// TwinCAT 3 PLC project Library
// Title: lcls-twincat-common-components
// Company: SLAC
// ProjectVersion: 0.0.0
// ProgramVersion: 3.1.4026.17
// libraries:
//   LCLS General, * (SLAC)
//   lcls-twincat-motion, * (SLAC)
//   lcls-twincat-physics, * (SLAC)
//   PMPS, * (SLAC - LCLS)
//   Tc2_MC2, * (Beckhoff Automation GmbH)
//   Tc2_SerialCom, * (Beckhoff Automation GmbH)
//   Tc2_Standard, * (Beckhoff Automation GmbH)
//   Tc2_System, * (Beckhoff Automation GmbH)
//   Tc2_Utilities, * (Beckhoff Automation GmbH)
//   Tc3_JsonXml, * (Beckhoff Automation GmbH)
//   Tc3_Module, * (Beckhoff Automation GmbH)
//   TcUnit, * (www.tcunit.org)
// project tree:
//   Devices/ATM/ E_ATM_States.TcDUT (not stored), FB_ATM.TcPOU (not stored)
//   Devices/HE_SATT/ E_HE_SATT_FilterMaterial.TcDUT, E_HE_SATT_FilterStatus.TcDUT, E_HE_SATT_FilterType.TcDUT, E_HE_SATT_RoundingMode.TcDUT, E_HE_SATT_SequenceState.TcDUT, F_HE_SATT_MaterialToMaterialFormula.TcPOU, PL_HE_SATT_Parameters.TcGVL, ST_HE_SATT_Status.TcDUT
//   Devices/HE_SATT/FBs/ FB_HE_SATT.TcPOU, FB_HE_SATT_CommandsEpics.TcPOU, FB_HE_SATT_EpicsHeartBeat.TcPOU, FB_HE_SATT_Filter.TcPOU, FB_HE_SATT_FilterCombination.TcPOU (not stored), FB_HE_SATT_FilterCombinationCollector.TcPOU, FB_HE_SATT_FilterCombinationFinder.TcPOU, FB_HE_SATT_FilterCombinationToTransmission.TcPOU, FB_HE_SATT_FilterConstantThickness.TcPOU, FB_HE_SATT_FilterHolder.TcPOU, FB_HE_SATT_FilterHolderSelector.TcPOU, FB_HE_SATT_FindOptimalFilterCombination.TcPOU, FB_HE_SATT_FilterToTransmission.TcPOU, FB_HE_SATT_FilterWedge.TcPOU, FB_HE_SATT_Sequence.TcPOU, FB_HE_SATT_UserRequest.TcPOU
//   Devices/HE_SATT/ITFs/ I_HE_SATT_Commands.TcIO, I_HE_SATT_Filter.TcIO, I_HE_SATT_FilterCombination.TcIO, I_HE_SATT_FilterCombinationCollector.TcIO, I_HE_SATT_FilterCombinationFinder.TcIO, I_HE_SATT_FilterCombinationToTransmission.TcIO, I_HE_SATT_FilterConstantThickness.TcIO (not stored), I_HE_SATT_FilterHolder.TcIO, I_HE_SATT_FilterHolderSelector.TcIO, I_HE_SATT_FilterToTransmission.TcIO, I_HE_SATT_FilterWedge.TcIO, I_HE_SATT_FindOptimalFilterCombination.TcIO, I_HE_SATT_FindOptimalThicknessFromFilterCombination.TcIO, I_HE_SATT_PhotonEnergy_eV.TcIO, I_HE_SATT_Sequence.TcIO
//   Devices/LIC/ E_LIC_States.TcDUT (not stored), FB_LIC.TcPOU (not stored)
//   Devices/PPM/ E_PPM_States.TcDUT (not stored), FB_PPM.TcPOU (not stored), FB_PPM_Gige.TcPOU (not stored), FB_PPM_PowerMeter.TcPOU
//   Devices/REF/ FB_REF.TcPOU (not stored), FB_REF_Laser.TcPOU (not stored)
//   Devices/SATT/ E_SXR_SATT_Position.TcDUT (not stored), FB_AttenuatorElementDensity.TcPOU (not stored), FB_SXR_SATT_Stage.TcPOU (not stored), ST_SATT_Filter.TcDUT (not stored)
//   Devices/SLITS/ FB_SLITS.TcPOU (not stored), FB_SLITS_POWER.TcPOU (not stored)
//   Devices/WFS/ E_WFS_States.TcDUT (not stored), FB_WFS.TcPOU (not stored)
//   Devices/GBS/ E_GBS_States.TcDUT (not stored), FB_GBS.TcPOU (not stored)
//   Devices/IPM/ E_IPM_States.TcDUT (not stored), FB_IPM.TcPOU (not stored)
//   Devices/XPIM/ E_XPIM_Filters.TcDUT (not stored), E_XPIM_States.TcDUT (not stored), FB_XPIM.TcPOU (not stored), FB_XPIM_FilterWheel.TcPOU (not stored), FB_XPIM_LED.TcPOU (not stored), FB_XPIM_Opal.TcPOU (not stored)
//   / PlcTask.TcTTO (not stored)
//   POUs/ FB_CC_TempSensor.TcPOU (not stored), FB_CheckPositionStateWrite.TcPOU (not stored), FB_FDQ_FlowMeter.TcPOU (not stored), FB_XTES_Flowswitch.TcPOU (not stored), FB_PositionState_Defaults.TcPOU (not stored)
//   Tests/ FB_ATMTest.TcPOU (not stored), FB_CC_TempSensorTest.TcPOU (not stored), FB_SATTTest.TcPOU (not stored), FB_CheckPositionStateWriteTest.TcPOU (not stored), FB_LICTest.TcPOU (not stored), FB_PPMTest.TcPOU (not stored), FB_REFTest.TcPOU (not stored), FB_SLITS_POWERTest.TcPOU (not stored), FB_WFSTest.TcPOU (not stored), FB_XPIMTest.TcPOU (not stored), PRG_TEST.TcPOU
//   Tests/Helpers/ FB_PMPSJsonTestHelper.TcPOU (not stored)
//   Tests/HE_SATT/ FB_HE_SATT_EpicsHeartBeat_Test.TcPOU, FB_HE_SATT_FilterCombinationCollector_Test.TcPOU, FB_HE_SATT_FindOptimalFilterCombination_Test.TcPOU, FB_HE_SATT_FilterHolderSelector_Test.TcPOU, FB_HE_SATT_FilterCombinationFinder_Test.TcPOU, FB_HE_SATT_FilterCombinationToTransmission_Test.TcPOU, FB_HE_SATT_FilterToTransmission_Test.TcPOU, FB_HE_SATT_UserRequest_Test.TcPOU
//   Tests/Test Doubles/ FB_HE_SATT_FilterCombinationToTransmissionTestDouble.TcPOU, FB_HE_SATT_FilterHolderSelectorTestDouble.TcPOU, FB_HE_SATT_FilterHolderTestDouble.TcPOU, FB_HE_SATT_FilterTestDouble.TcPOU, FB_HE_SATT_SequenceTestDouble.TcPOU
//   Version/ Global_Version.TcGVL (not stored)
// real-time tasks:
//   TASK PlcTask: cycle T#10ms, priority 20, ADS port 350
// motion (NC):

// ---- Devices/HE_SATT/E_HE_SATT_FilterMaterial.TcDUT
{attribute 'qualified_only'}
{attribute 'strict'}
{attribute 'to_string'}
TYPE E_HE_SATT_FilterMaterial :
(
    Silicon := 0,
    Diamond,
    Germanium
);
END_TYPE

// ---- Devices/HE_SATT/E_HE_SATT_FilterStatus.TcDUT
{attribute 'qualified_only'}
{attribute 'strict'}
{attribute 'to_string'}
TYPE E_HE_SATT_FilterStatus :
(
	DISABLED := 0,
    ENABLED
);
END_TYPE

// ---- Devices/HE_SATT/E_HE_SATT_FilterType.TcDUT
{attribute 'qualified_only'}
{attribute 'strict'}
{attribute 'to_string'}
TYPE E_HE_SATT_FilterType :
(
    None := 0,
    FixedThickness,
    Wedge
);
END_TYPE

// ---- Devices/HE_SATT/E_HE_SATT_RoundingMode.TcDUT
{attribute 'qualified_only'}
{attribute 'strict'}
{attribute 'to_string'}
TYPE E_HE_SATT_RoundingMode :
(
    FIRST_BELOW_WITHIN_TOLERANCE := 0,
    CLOSEST_ABOVE,
    CLOSEST_BELOW,
    CLOSEST,
    FIRST_ABOVE_WITHIN_TOLERANCE,
    FIRST_WITHIN_TOLERANCE
) UINT;
END_TYPE

// ---- Devices/HE_SATT/E_HE_SATT_SequenceState.TcDUT
{attribute 'qualified_only'}
{attribute 'strict'}
{attribute 'to_string'}
TYPE E_HE_SATT_SequenceState :
(
    IDLE := 0,
    ERROR,
    TRIGGER_DETERMINE_FILTER_COMBINATIONS,
    CONFIRM_DETERMINE_FILTER_COMBINATIONS,
    TRIGGER_DOWNSELECT_FILTER_COMBINATIONS,
    CONFIRM_DOWNSELECT_FILTER_COMBINATIONS,
    TRIGGER_CALCULATE_OPTIMAL_FILTER_COMBINATION,
    CONFIRM_CALCULATE_OPTIMAL_FILTER_COMBINATION,
    TRIGGER_CALCULATE_OPTIMAL_WEDGE_THICKNESSES,
    CONFIRM_CALCULATE_OPTIMAL_WEDGE_THICKNESSES,
    CONFIRM_MOVE_PERMITTED,
    TRIGGER_MOVE_START,
    CONFIRM_MOVE_COMPLETE
);
END_TYPE

// ---- Devices/HE_SATT/ST_HE_SATT_Status.TcDUT

TYPE ST_HE_SATT_Status :
STRUCT
    bBusy : BOOL;
    bDone : BOOL;
    bError : BOOL;
    sErrorMsg : T_MaxString;
END_STRUCT
END_TYPE

// ---- Devices/HE_SATT/PL_HE_SATT_Parameters.TcGVL
{attribute 'qualified_only'}
VAR_GLOBAL CONSTANT
    nNumHolders : INT := 5;
    nMaxNumFiltersPerHolder : INT := 11;
END_VAR

// ---- Devices/HE_SATT/ITFs/I_HE_SATT_Commands.TcIO

INTERFACE I_HE_SATT_Commands


PROPERTY PermitMove : BOOL
GET
END_GET
END_PROPERTY


PROPERTY Reset : BOOL
GET
END_GET
END_PROPERTY

END_INTERFACE

// ---- Devices/HE_SATT/ITFs/I_HE_SATT_Filter.TcIO

INTERFACE I_HE_SATT_Filter EXTENDS __System.IQueryInterface


PROPERTY Holder : I_HE_SATT_FilterHolder
GET
END_GET
END_PROPERTY


PROPERTY Length : LREAL
GET
END_GET
END_PROPERTY


PROPERTY Material : E_HE_SATT_FilterMaterial
GET
END_GET
END_PROPERTY

PROPERTY MaterialFormula : T_MaxString
GET
END_GET
END_PROPERTY

PROPERTY Status : E_HE_SATT_FilterStatus
GET
END_GET
END_PROPERTY

END_INTERFACE

// ---- Devices/HE_SATT/ITFs/I_HE_SATT_FilterCombination.TcIO

INTERFACE I_HE_SATT_FilterCombination


METHOD AddFilter
VAR_INPUT
    nHolderNumber : INT;
    iFilter : I_HE_SATT_Filter;
END_VAR
END_METHOD


METHOD Clear
END_METHOD


METHOD GetFilter : I_HE_SATT_Filter
VAR_INPUT
    nHolderNumber : INT;
END_VAR
END_METHOD

PROPERTY HolderNumberOfLastFilterAdded : INT
GET
END_GET
END_PROPERTY


METHOD PUBLIC IsValidHolderNumber : BOOL
VAR_INPUT
    nHolderNumber : INT;
END_VAR
END_METHOD


METHOD RemoveFilter
VAR_INPUT
    nHolderNumber : INT;
END_VAR
END_METHOD

END_INTERFACE

// ---- Devices/HE_SATT/ITFs/I_HE_SATT_FilterCombinationCollector.TcIO

INTERFACE I_HE_SATT_FilterCombinationCollector


METHOD PUBLIC AddFilterCombination
VAR_INPUT
    fbFilterCombination : REFERENCE TO FB_HE_SATT_FilterCombination;
END_VAR
END_METHOD


METHOD PUBLIC DownselectByCouplingRule
VAR_INPUT
    iFilterCombinationCollector : I_HE_SATT_FilterCombinationCollector;
    iFilterHolderSelector : I_HE_SATT_FilterHolderSelector;
END_VAR
END_METHOD


PROPERTY DownselectStatus : REFERENCE TO ST_HE_SATT_Status
GET
END_GET
END_PROPERTY


METHOD GetCombination : REFERENCE TO FB_HE_SATT_FilterCombination
VAR_INPUT
    nCombinationNumber : DINT;
END_VAR
END_METHOD


PROPERTY NumCombinationsAdded : DINT
GET
END_GET
END_PROPERTY


METHOD PUBLIC Reset
END_METHOD

END_INTERFACE

// ---- Devices/HE_SATT/ITFs/I_HE_SATT_FilterCombinationFinder.TcIO

INTERFACE I_HE_SATT_FilterCombinationFinder


METHOD PUBLIC DetermineFilterCombinations
VAR_INPUT
    iFilterHolderSelector : I_HE_SATT_FilterHolderSelector;
    iFilterCombinationCollector : I_HE_SATT_FilterCombinationCollector;
END_VAR
END_METHOD


PROPERTY Status : REFERENCE TO ST_HE_SATT_Status
GET
END_GET
END_PROPERTY

END_INTERFACE

// ---- Devices/HE_SATT/ITFs/I_HE_SATT_FilterCombinationToTransmission.TcIO
INTERFACE I_HE_SATT_FilterCombinationToTransmission


METHOD PUBLIC CalculateTransmission
VAR_INPUT
    fPhotonEnergy_eV : LREAL;
    iFilterCombination : I_HE_SATT_FilterCombination;
END_VAR
VAR_OUTPUT
    fMinimumTransmission : LREAL;
    fMaximumTransmission : LREAL;
END_VAR
END_METHOD

END_INTERFACE

// ---- Devices/HE_SATT/ITFs/I_HE_SATT_FilterHolder.TcIO

INTERFACE I_HE_SATT_FilterHolder


METHOD GetFilter : I_HE_SATT_Filter
VAR_INPUT
    nFilterNumber : INT;
END_VAR
END_METHOD


METHOD MoveToFilter
VAR_INPUT
    iFilter : I_HE_SATT_Filter;
    fThickness : LREAL;
END_VAR
END_METHOD


PROPERTY NumberOfSlots : INT
GET
END_GET
END_PROPERTY


METHOD RegisterFilter
VAR_INPUT
    iFilter : I_HE_SATT_Filter;
END_VAR
END_METHOD


PROPERTY Status : REFERENCE TO ST_HE_SATT_Status
GET
END_GET
END_PROPERTY

END_INTERFACE

// ---- Devices/HE_SATT/ITFs/I_HE_SATT_FilterHolderSelector.TcIO
INTERFACE I_HE_SATT_FilterHolderSelector


METHOD CoupleHolders
VAR_INPUT
    abCoupledHolders : ARRAY[1..PL_HE_SATT_Parameters.nNumHolders] OF BOOL;
END_VAR
END_METHOD


METHOD CouplingRulesSatisfied : BOOL
VAR_INPUT
    iFilterCombination : I_HE_SATT_FilterCombination;
END_VAR
END_METHOD


METHOD DeselectHolder
VAR_INPUT
    nHolderNumber : INT;
END_VAR
END_METHOD


METHOD IsSelected : BOOL
VAR_INPUT
    nHolderNumber : INT;
END_VAR
END_METHOD


METHOD Reset
END_METHOD


METHOD SelectAll
END_METHOD


METHOD SelectHolder
VAR_INPUT
    nHolderNumber : INT;
END_VAR
END_METHOD

END_INTERFACE

// ---- Devices/HE_SATT/ITFs/I_HE_SATT_FilterToTransmission.TcIO
INTERFACE I_HE_SATT_FilterToTransmission


METHOD PUBLIC CalculateTransmission
VAR_INPUT
    fPhotonEnergy_eV : LREAL;
    iFilter : I_HE_SATT_Filter;
END_VAR
VAR_OUTPUT
    fMinimumTransmission : LREAL;
    fMaximumTransmission : LREAL;
END_VAR
END_METHOD

END_INTERFACE

// ---- Devices/HE_SATT/ITFs/I_HE_SATT_FilterWedge.TcIO

INTERFACE I_HE_SATT_FilterWedge EXTENDS I_HE_SATT_Filter

PROPERTY MaxThickness : LREAL
GET
END_GET
END_PROPERTY

PROPERTY MinThickness : LREAL
GET
END_GET
END_PROPERTY


METHOD ThicknessAt : LREAL
VAR_INPUT
    fPosition : LREAL; // Position in units of property Length and with value from 0 to value of property Length
END_VAR
END_METHOD

END_INTERFACE

// ---- Devices/HE_SATT/ITFs/I_HE_SATT_FindOptimalFilterCombination.TcIO

INTERFACE I_HE_SATT_FindOptimalFilterCombination


METHOD PUBLIC FindOptimalCombination
VAR_INPUT
    fPhotonEnergy_eV : LREAL;
	(* [0.0 - 1.0]*)
	fRequestedTransmission	: LREAL;
	eRequestedRoundingMode	: E_HE_SATT_RoundingMode;
	fRequestedAllowableTolerance	: LREAL;
    iFilterCombinationCollector : I_HE_SATT_FilterCombinationCollector;
END_VAR
VAR_OUTPUT
    iOptimalFilterCombination : I_HE_SATT_FilterCombination;
END_VAR
END_METHOD


PROPERTY Status : REFERENCE TO ST_HE_SATT_Status
GET
END_GET
END_PROPERTY

END_INTERFACE

// ---- Devices/HE_SATT/ITFs/I_HE_SATT_FindOptimalThicknessFromFilterCombination.TcIO

INTERFACE I_HE_SATT_FindOptimalThicknessFromFilterCombination


METHOD FindOptimalThicknessFromFilterCombination
VAR_INPUT
    fPhotonEnergy_eV : LREAL;
    fRequestedTransmission : LREAL;
    iFilterCombination : I_HE_SATT_FilterCombination;
END_VAR
VAR_OUTPUT
    afThickness : ARRAY[1..PL_HE_SATT_Parameters.nNumHolders] OF LREAL;
END_VAR
END_METHOD


PROPERTY Status : REFERENCE TO ST_HE_SATT_Status
GET
END_GET
END_PROPERTY

END_INTERFACE

// ---- Devices/HE_SATT/ITFs/I_HE_SATT_PhotonEnergy_eV.TcIO

INTERFACE I_HE_SATT_PhotonEnergy_eV


PROPERTY Error : BOOL
GET
END_GET
END_PROPERTY


PROPERTY Value : LREAL
GET
END_GET
END_PROPERTY

END_INTERFACE

// ---- Devices/HE_SATT/ITFs/I_HE_SATT_Sequence.TcIO
INTERFACE I_HE_SATT_Sequence


METHOD Start
VAR_INPUT
    fRequestedTransmission : LREAL; // [0.0 - 1.0]
    eRequestedRoundingMode : E_HE_SATT_RoundingMode;
    fRequestedAllowableTolerance : LREAL;
END_VAR
END_METHOD

END_INTERFACE

// ---- Devices/HE_SATT/FBs/FB_HE_SATT.TcPOU

FUNCTION_BLOCK FB_HE_SATT
VAR
END_VAR


METHOD CallAfterInit
END_METHOD

END_FUNCTION_BLOCK

// ---- Devices/HE_SATT/FBs/FB_HE_SATT_CommandsEpics.TcPOU

FUNCTION_BLOCK FB_HE_SATT_CommandsEpics IMPLEMENTS I_HE_SATT_Commands
VAR
    bPermitMove : BOOL;
    bReset : BOOL;
END_VAR


PROPERTY PermitMove : BOOL
GET

PermitMove := THIS^.bPermitMove;
END_GET
SET

THIS^.bPermitMove := PermitMove;
END_SET
END_PROPERTY


PROPERTY Reset : BOOL
GET

Reset := THIS^.bReset;
END_GET
SET

THIS^.bReset := Reset;
END_SET
END_PROPERTY

END_FUNCTION_BLOCK

// ---- Devices/HE_SATT/FBs/FB_HE_SATT_EpicsHeartBeat.TcPOU
FUNCTION_BLOCK FB_HE_SATT_EpicsHeartBeat
VAR
    bHeartbeat : BOOL; // TRUE needs to be written to this externally
    fbHeartbeatTimer : TON;
END_VAR


fbHeartbeatTimer(IN := NOT bHeartbeat);
bHeartbeat := FALSE;

//FB_Init is always available implicitly and it is used primarily for initialization.
//The return value is not evaluated. For a specific influence, you can also declare the
//methods explicitly and provide additional code there with the standard initialization
//code. You can evaluate the return value.
METHOD FB_Init: BOOL
VAR_INPUT
    bInitRetains: BOOL; // TRUE: the retain variables are initialized (reset warm / reset cold)
    bInCopyCode: BOOL;  // TRUE: the instance will be copied to the copy code afterward (online change)
    tTimeout : TIME;
END_VAR
fbHeartbeatTimer.PT := tTimeout;
END_METHOD

METHOD PUBLIC Heartbeat
THIS^.bHeartbeat := TRUE;
END_METHOD

METHOD PUBLIC IsHeartbeatExpired : BOOL

IsHeartbeatExpired := THIS^.fbHeartbeatTimer.Q;
END_METHOD

END_FUNCTION_BLOCK

// ---- Devices/HE_SATT/FBs/FB_HE_SATT_Filter.TcPOU

FUNCTION_BLOCK ABSTRACT FB_HE_SATT_Filter IMPLEMENTS I_HE_SATT_Filter
VAR
    iHolder : I_HE_SATT_FilterHolder;
    fLength : LREAL;
    eMaterial : E_HE_SATT_FilterMaterial;
    eStatus : E_HE_SATT_FilterStatus;
END_VAR


METHOD FB_Init: BOOL
VAR_INPUT
    bInitRetains: BOOL; // TRUE: the retain variables are initialized (reset warm / reset cold)
    bInCopyCode: BOOL;  // TRUE: the instance will be copied to the copy code afterward (online change)   
    
    iHolder : I_HE_SATT_FilterHolder;
    fDefaultLength : LREAL;
    eDefaultMaterial : E_HE_SATT_FilterMaterial;
    eDefaultStatus : E_HE_SATT_FilterStatus;
END_VAR

THIS^.iHolder := iHolder;
THIS^.fLength := fDefaultLength;
THIS^.eMaterial := eDefaultMaterial;
THIS^.eStatus := eDefaultStatus;
END_METHOD


PROPERTY Holder : I_HE_SATT_FilterHolder
GET

Holder := THIS^.iHolder;
END_GET
END_PROPERTY


PROPERTY Length : LREAL
GET

Length := THIS^.fLength;
END_GET
SET

THIS^.fLength := Length;
END_SET
END_PROPERTY


PROPERTY Material : E_HE_SATT_FilterMaterial
GET

Material := THIS^.eMaterial;
END_GET
SET

THIS^.eMaterial := Material;
END_SET
END_PROPERTY


PROPERTY MaterialFormula : T_MaxString
GET

MaterialFormula := F_HE_SATT_MaterialToMaterialFormula(eMaterial := THIS^.eMaterial);
END_GET
END_PROPERTY


PROPERTY Status : E_HE_SATT_FilterStatus
GET

Status := THIS^.eStatus;
END_GET
SET

THIS^.eStatus := Status;
END_SET
END_PROPERTY

END_FUNCTION_BLOCK

// ---- Devices/HE_SATT/F_HE_SATT_MaterialToMaterialFormula.TcPOU

FUNCTION F_HE_SATT_MaterialToMaterialFormula : T_MaxString
VAR_INPUT
    eMaterial : E_HE_SATT_FilterMaterial;
END_VAR


CASE eMaterial OF
    E_HE_SATT_FilterMaterial.Diamond:
        F_HE_SATT_MaterialToMaterialFormula := 'C (Diamond)';
        
    E_HE_SATT_FilterMaterial.Germanium:
        F_HE_SATT_MaterialToMaterialFormula := 'Ge';
        
    E_HE_SATT_FilterMaterial.Silicon:
        F_HE_SATT_MaterialToMaterialFormula := 'Si';
        
    ELSE
        F_HE_SATT_MaterialToMaterialFormula := TO_STRING(eMaterial);
END_CASE

END_FUNCTION

// ---- Devices/HE_SATT/FBs/FB_HE_SATT_FilterCombinationCollector.TcPOU

FUNCTION_BLOCK FB_HE_SATT_FilterCombinationCollector IMPLEMENTS I_HE_SATT_FilterCombinationCollector
VAR CONSTANT
    nMAXIMUM_NUMBER_OF_COMBINATIONS : DINT := 1000;
END_VAR
VAR
    nNumberOfCombinations : DINT;
    afbFilterCombination : ARRAY[1..nMAXIMUM_NUMBER_OF_COMBINATIONS] OF FB_HE_SATT_FilterCombination;
    stStatus : ST_HE_SATT_Status;
    eState : (DOWNSELECTING, IDLE);
    
    nCombinationIterator : DINT;
    nNumCombinationsAdded : DINT;
    fbFilterCombination : REFERENCE TO FB_HE_SATT_FilterCombination;
    iFilterCombinationCollector : I_HE_SATT_FilterCombinationCollector;
    iFilterHolderSelector : I_HE_SATT_FilterHolderSelector;
END_VAR


CASE eState OF
    IDLE:
        stStatus.bBusy := FALSE;
        
    DOWNSELECTING:
        stStatus.bBusy := TRUE;
        
        nNumCombinationsAdded := THIS^.NumCombinationsAdded;
        
        FOR nCombinationIterator := 1 TO nNumCombinationsAdded BY 1 DO
            fbFilterCombination REF= THIS^.GetCombination(nCombinationIterator);
            
            IF NOT __ISVALIDREF(fbFilterCombination) OR_ELSE NOT iFilterHolderSelector.CouplingRulesSatisfied(fbFilterCombination) THEN
                CONTINUE;
            END_IF
            
            iFilterCombinationCollector.AddFilterCombination(fbFilterCombination);
        END_FOR
        
        stStatus.bBusy := FALSE;
        stStatus.bDone := TRUE;
        stStatus.bError := FALSE;
        stStatus.sErrorMsg := '';
        
        eState := IDLE;
END_CASE


METHOD PUBLIC AddFilterCombination
VAR_INPUT
    fbFilterCombination : REFERENCE TO FB_HE_SATT_FilterCombination;
END_VAR

IF nNumberOfCombinations >= nMAXIMUM_NUMBER_OF_COMBINATIONS THEN
    RETURN;
END_IF

nNumberOfCombinations := nNumberOfCombinations + 1;
afbFilterCombination[nNumberOfCombinations] := fbFilterCombination;
END_METHOD


METHOD PUBLIC DownselectByCouplingRule
VAR_INPUT
    iFilterCombinationCollector : I_HE_SATT_FilterCombinationCollector;
    iFilterHolderSelector : I_HE_SATT_FilterHolderSelector;
END_VAR

THIS^.iFilterCombinationCollector := iFilterCombinationCollector;
THIS^.iFilterHolderSelector := iFilterHolderSelector;

THIS^.stStatus.bBusy := TRUE;
THIS^.stStatus.bDone := FALSE;
THIS^.stStatus.bError := FALSE;
THIS^.stStatus.sErrorMsg := '';

THIS^.eState := DOWNSELECTING;
END_METHOD


PROPERTY DownselectStatus : REFERENCE TO ST_HE_SATT_Status
GET

DownselectStatus REF= THIS^.stStatus;
END_GET
END_PROPERTY


METHOD GetCombination : REFERENCE TO FB_HE_SATT_FilterCombination
VAR_INPUT
	nCombinationNumber	: DINT;
END_VAR

GetCombination REF= afbFilterCombination[nCombinationNumber];
END_METHOD


PROPERTY NumCombinationsAdded : DINT
GET

NumCombinationsAdded := THIS^.nNumberOfCombinations;
END_GET
END_PROPERTY


METHOD PUBLIC Reset

nNumberOfCombinations := 0;
END_METHOD

END_FUNCTION_BLOCK

// ---- Devices/HE_SATT/FBs/FB_HE_SATT_FilterCombinationFinder.TcPOU

FUNCTION_BLOCK FB_HE_SATT_FilterCombinationFinder IMPLEMENTS I_HE_SATT_FilterCombinationFinder
VAR
    aiFilterHolder : REFERENCE TO ARRAY[1..PL_HE_SATT_Parameters.nNumHolders] OF I_HE_SATT_FilterHolder;
    iFilterCombinationCollector : I_HE_SATT_FilterCombinationCollector;
    nMaxNumberOfCombinationsFoundPerCycle : INT;
    
    eState : (IDLE, FINDING_COMBINATIONS);
    
    iFilterHolderSelector : I_HE_SATT_FilterHolderSelector;
    
    stStatus : ST_HE_SATT_Status;
    
    nFilterHolderIterator : INT; 
    nFilterHolderIteratorLastCycle : INT;
    
    nCombinationIterator : DINT;
    nCombinationIteratorLastCycle : DINT;
    
    nNumCombinationsThusFar : DINT;  
    
    nFilterIterator : INT;   
    nFilterIteratorLastCycle : INT; 
    
    nMaxNumberOfCombinationsForThisCycle : DINT;
    
    iFilter : I_HE_SATT_Filter;

    fbFilterCombination : FB_HE_SATT_FilterCombination;
END_VAR


CASE eState OF
    IDLE:
        stStatus.bBusy := FALSE;
        
    FINDING_COMBINATIONS:
        
        FOR nFilterHolderIterator := nFilterHolderIteratorLastCycle TO PL_HE_SATT_Parameters.nNumHolders BY 1 DO
            IF NOT iFilterHolderSelector.IsSelected(nFilterHolderIterator) THEN
                CONTINUE;
            END_IF
            
            FOR nCombinationIterator := nCombinationIteratorLastCycle TO nNumCombinationsThusFar BY 1 DO
                FOR nFilterIterator := nFilterIteratorLastCycle + 1 TO aiFilterHolder[nFilterHolderIterator].NumberOfSlots BY 1 DO
                    fbFilterCombination := iFilterCombinationCollector.GetCombination(
                        nCombinationNumber := nCombinationIterator
                    );
                    
                    iFilter := aiFilterHolder[nFilterHolderIterator].GetFilter(
                        nFilterNumber := nFilterIterator
                    );
                    
                    IF iFilter.Status = E_HE_SATT_FilterStatus.DISABLED THEN
                        CONTINUE;
                    END_IF
                    
                    fbFilterCombination.AddFilter(
                        nHolderNumber := nFilterHolderIterator,
                        iFilter := iFilter
                    );
                    
                    iFilterCombinationCollector.AddFilterCombination(
                        fbFilterCombination := fbFilterCombination
                    );
                        
                    IF iFilterCombinationCollector.NumCombinationsAdded < nMaxNumberOfCombinationsForThisCycle THEN
                        CONTINUE;
                    END_IF
                    
                    nFilterHolderIteratorLastCycle := nFilterHolderIterator;
                    nCombinationIteratorLastCycle := nCombinationIterator;
                    nFilterIteratorLastCycle := nFilterIterator;
                    nMaxNumberOfCombinationsForThisCycle := nMaxNumberOfCombinationsForThisCycle + nMaxNumberOfCombinationsFoundPerCycle;
                    RETURN;
                END_FOR
            END_FOR
            nNumCombinationsThusFar := iFilterCombinationCollector.NumCombinationsAdded; 
        END_FOR
        
        stStatus.bBusy := FALSE;
        stStatus.bDone := TRUE;
        stStatus.bError := FALSE;
        stStatus.sErrorMsg := '';
        
        eState := IDLE;
END_CASE


METHOD PUBLIC DetermineFilterCombinations
VAR_INPUT
    iFilterHolderSelector : I_HE_SATT_FilterHolderSelector;
    iFilterCombinationCollector : I_HE_SATT_FilterCombinationCollector;
END_VAR

THIS^.iFilterHolderSelector := iFilterHolderSelector;

THIS^.iFilterCombinationCollector := iFilterCombinationCollector;
    
THIS^.stStatus.bBusy := TRUE;
THIS^.stStatus.bDone := FALSE;
THIS^.stStatus.bError := FALSE;
THIS^.stStatus.sErrorMsg := '';

THIS^.iFilterCombinationCollector.Reset();

THIS^.fbFilterCombination.Clear();

// First combination that is always valid is the combination which doesn't use any filters.
THIS^.iFilterCombinationCollector.AddFilterCombination(
    fbFilterCombination := THIS^.fbFilterCombination
);

THIS^.nFilterHolderIteratorLastCycle := 1;
THIS^.nCombinationIteratorLastCycle := 1;
THIS^.nFilterIteratorLastCycle := 0;

THIS^.nNumCombinationsThusFar := THIS^.iFilterCombinationCollector.NumCombinationsAdded;

THIS^.nMaxNumberOfCombinationsForThisCycle := THIS^.nMaxNumberOfCombinationsFoundPerCycle;

THIS^.eState := FINDING_COMBINATIONS;
END_METHOD


METHOD FB_Init: BOOL
VAR_INPUT
    bInitRetains: BOOL; // TRUE: the retain variables are initialized (reset warm / reset cold)
    bInCopyCode: BOOL;  // TRUE: the instance will be copied to the copy code afterward (online change)
    
    aiFilterHolder : REFERENCE TO ARRAY[1..PL_HE_SATT_Parameters.nNumHolders] OF I_HE_SATT_FilterHolder;
    nMaxNumberOfCombinationsFoundPerCycle : INT;
END_VAR

THIS^.aiFilterHolder REF= aiFilterHolder;
THIS^.nMaxNumberOfCombinationsFoundPerCycle := nMaxNumberOfCombinationsFoundPerCycle;
END_METHOD


PROPERTY Status : REFERENCE TO ST_HE_SATT_Status
GET

Status REF= THIS^.stStatus;
END_GET
END_PROPERTY

END_FUNCTION_BLOCK

// ---- Devices/HE_SATT/FBs/FB_HE_SATT_FilterCombinationToTransmission.TcPOU

FUNCTION_BLOCK FB_HE_SATT_FilterCombinationToTransmission
VAR
    iFilterToTransmission : I_HE_SATT_FilterToTransmission;
END_VAR


METHOD PUBLIC CalculateTransmission
VAR_INPUT
    fPhotonEnergy_eV : LREAL;
    iFilterCombination : I_HE_SATT_FilterCombination;
END_VAR
VAR_OUTPUT
    fMinimumTransmission : LREAL;
    fMaximumTransmission : LREAL;
END_VAR
VAR
    nIteratorHolder : INT;
    iFilter : I_HE_SATT_Filter;
    fMinimumTransmissionTemp : LREAL;
    fMaximumTransmissionTemp : LREAL;
END_VAR

fMinimumTransmission := 1.0;
fMaximumTransmission := 1.0;

FOR nIteratorHolder := 1 TO PL_HE_SATT_Parameters.nNumHolders BY 1 DO
    iFilter := iFilterCombination.GetFilter(nIteratorHolder);
    
    IF iFilter = 0 THEN
        CONTINUE;
    END_IF
    
    THIS^.iFilterToTransmission.CalculateTransmission(
        fPhotonEnergy_eV := fPhotonEnergy_eV,
        iFilter := iFilter,
        fMinimumTransmission => fMinimumTransmissionTemp,
        fMaximumTransmission => fMaximumTransmissionTemp
    );
    
    fMinimumTransmission := fMinimumTransmission * fMinimumTransmissionTemp;
    fMaximumTransmission := fMaximumTransmission * fMaximumTransmissionTemp;
END_FOR
END_METHOD


METHOD FB_Init: BOOL
VAR_INPUT
    bInitRetains: BOOL; // TRUE: the retain variables are initialized (reset warm / reset cold)
    bInCopyCode: BOOL;  // TRUE: the instance will be copied to the copy code afterward (online change)   
    
    iFilterToTransmission : I_HE_SATT_FilterToTransmission;
END_VAR

THIS^.iFilterToTransmission := iFilterToTransmission;
END_METHOD

END_FUNCTION_BLOCK

// ---- Devices/HE_SATT/FBs/FB_HE_SATT_FilterConstantThickness.TcPOU

FUNCTION_BLOCK FB_HE_SATT_FilterConstantThickness EXTENDS FB_HE_SATT_Filter IMPLEMENTS I_HE_SATT_FilterConstantThickness
VAR
    fThickness : LREAL;
END_VAR


METHOD FB_Init: BOOL
VAR_INPUT
    bInitRetains: BOOL; // TRUE: the retain variables are initialized (reset warm / reset cold)
    bInCopyCode: BOOL;  // TRUE: the instance will be copied to the copy code afterward (online change)   
    
    iHolder : I_HE_SATT_FilterHolder;
    fDefaultLength : LREAL;
    eDefaultMaterial : E_HE_SATT_FilterMaterial;
    eDefaultStatus : E_HE_SATT_FilterStatus;
    fDefaultThickness : LREAL;
END_VAR

THIS^.iHolder := iHolder;
THIS^.fLength := fDefaultLength;
THIS^.eMaterial := eDefaultMaterial;
THIS^.eStatus := eDefaultStatus;
THIS^.fThickness := fDefaultThickness;

THIS^.iHolder.RegisterFilter(THIS^);
END_METHOD


PROPERTY Thickness : LREAL
GET

Thickness := THIS^.fThickness;
END_GET
SET

THIS^.fThickness := Thickness;
END_SET
END_PROPERTY

END_FUNCTION_BLOCK

// ---- Devices/HE_SATT/FBs/FB_HE_SATT_FilterHolder.TcPOU

FUNCTION_BLOCK FB_HE_SATT_FilterHolder IMPLEMENTS I_HE_SATT_FilterHolder
VAR
END_VAR


METHOD FB_Init: BOOL
VAR_INPUT
    bInitRetains: BOOL; // TRUE: the retain variables are initialized (reset warm / reset cold)
    bInCopyCode: BOOL;  // TRUE: the instance will be copied to the copy code afterward (online change)

//     iMotionStage : I_MotionStage;  
END_VAR
END_METHOD

{warning 'Add method implementation '}
METHOD GetFilter : I_HE_SATT_Filter
VAR_INPUT
	nFilterNumber	: INT;
END_VAR
END_METHOD


METHOD MoveToFilter
VAR_INPUT
    iFilter : I_HE_SATT_Filter;
    fThickness : LREAL;
END_VAR
END_METHOD

{warning 'Add property implementation'}
PROPERTY NumberOfSlots : INT
GET
END_GET
END_PROPERTY

{warning 'Add method implementation '}
METHOD RegisterFilter
VAR_INPUT
	iFilter	: I_HE_SATT_Filter;
END_VAR
END_METHOD

{warning 'Add property implementation'}
PROPERTY Status : REFERENCE TO ST_HE_SATT_Status
GET
END_GET
END_PROPERTY

END_FUNCTION_BLOCK

// ---- Devices/HE_SATT/FBs/FB_HE_SATT_FilterHolderSelector.TcPOU

FUNCTION_BLOCK FB_HE_SATT_FilterHolderSelector IMPLEMENTS I_HE_SATT_FilterHolderSelector
VAR
    abSelectedHolder : ARRAY[1..PL_HE_SATT_Parameters.nNumHolders] OF BOOL;
    abCoupledHolders : ARRAY[1..PL_HE_SATT_Parameters.nNumHolders] OF BOOL;
END_VAR


METHOD CoupleHolders
VAR_INPUT
	abCoupledHolders : ARRAY [1..PL_HE_SATT_Parameters.nNumHolders] OF BOOL;
END_VAR

THIS^.abCoupledHolders := abCoupledHolders;
END_METHOD


METHOD CouplingRulesSatisfied : BOOL
VAR_INPUT
	iFilterCombination	: I_HE_SATT_FilterCombination;
END_VAR
VAR
    abFilterHolderIsUsed : ARRAY[1..PL_HE_SATT_Parameters.nNumHolders] OF BOOL;
    nIteratorHolder : INT;
    iFilter : I_HE_SATT_Filter;
    bStateAllCoupledHoldersNeedToBeIn : BOOL;
END_VAR

CouplingRulesSatisfied := TRUE;

FOR nIteratorHolder := 1 TO PL_HE_SATT_Parameters.nNumHolders BY 1 DO
    iFilter := iFilterCombination.GetFilter(nIteratorHolder);
    
    abFilterHolderIsUsed[nIteratorHolder] := iFilter <> 0;
    
    IF THIS^.abCoupledHolders[nIteratorHolder] THEN
        bStateAllCoupledHoldersNeedToBeIn := abFilterHolderIsUsed[nIteratorHolder];
    END_IF
END_FOR

FOR nIteratorHolder := 1 TO PL_HE_SATT_Parameters.nNumHolders BY 1 DO
    IF THIS^.abCoupledHolders[nIteratorHolder] THEN
        CouplingRulesSatisfied := CouplingRulesSatisfied AND (NOT bStateAllCoupledHoldersNeedToBeIn XOR abFilterHolderIsUsed[nIteratorHolder]);
    END_IF
END_FOR
END_METHOD


METHOD DeselectHolder
VAR_INPUT
	nHolderNumber	: INT;
END_VAR

THIS^.abSelectedHolder[nHolderNumber] := FALSE;
END_METHOD


METHOD IsSelected : BOOL
VAR_INPUT
	nHolderNumber	: INT;
END_VAR

IsSelected := THIS^.abSelectedHolder[nHolderNumber];
END_METHOD


METHOD Reset
VAR
    nIteratorHolder : INT;
END_VAR

FOR nIteratorHolder := 1 TO PL_HE_SATT_Parameters.nNumHolders BY 1 DO
    THIS^.abSelectedHolder[nIteratorHolder] := FALSE;
END_FOR
END_METHOD

{warning 'Add method implementation '}
METHOD SelectAll
END_METHOD


METHOD SelectHolder
VAR_INPUT
	nHolderNumber	: INT;
END_VAR

THIS^.abSelectedHolder[nHolderNumber] := TRUE;
END_METHOD

END_FUNCTION_BLOCK

// ---- Devices/HE_SATT/FBs/FB_HE_SATT_FindOptimalFilterCombination.TcPOU

FUNCTION_BLOCK FB_HE_SATT_FindOptimalFilterCombination IMPLEMENTS I_HE_SATT_FindOptimalFilterCombination
VAR
    iFilterCombinationToTransmission : I_HE_SATT_FilterCombinationToTransmission;
    
    stStatus : ST_HE_SATT_Status;
    
    eState : (IDLE, FINDING_COMBINATIONS);
    
    fPhotonEnergy_eV : LREAL;
	(* [0.0 - 1.0]*)
	fRequestedTransmission	: LREAL;
	eRequestedRoundingMode	: E_HE_SATT_RoundingMode;
	fRequestedAllowableTolerance	: LREAL;
    iFilterCombinationCollector : I_HE_SATT_FilterCombinationCollector;
    
    iOptimalFilterCombination : I_HE_SATT_FilterCombination;
    
    nCombinationIterator : DINT;
    fbFilterCombination : REFERENCE TO FB_HE_SATT_FilterCombination;
    fMinimumTransmission : LREAL;
    fMaximumTransmission : LREAL;
    fAverageTransmission : LREAL;
    fOptimalAverageTransmissionThusFar : LREAL;
    fTransmissionError : LREAL;
    fOptimalTransmissionErrorThusFar : LREAL;
END_VAR


CASE eState OF
    IDLE:
        stStatus.bBusy := FALSE;
        
    FINDING_COMBINATIONS:
        stStatus.bBusy := TRUE;
        
        fOptimalTransmissionErrorThusFar := 10000.0;
        fOptimalAverageTransmissionThusFar := 10000.0;
        
        FOR nCombinationIterator := 1 TO iFilterCombinationCollector.NumCombinationsAdded DO
            fbFilterCombination REF= iFilterCombinationCollector.GetCombination(nCombinationIterator);
            
            THIS^.iFilterCombinationToTransmission.CalculateTransmission(
                fPhotonEnergy_eV :=  fPhotonEnergy_eV,
                iFilterCombination := fbFilterCombination,
                fMinimumTransmission => fMinimumTransmission,
                fMaximumTransmission => fMaximumTransmission
            );
            
            CASE eRequestedRoundingMode OF
                E_HE_SATT_RoundingMode.CLOSEST_ABOVE:
                    IF fRequestedTransmission > fMaximumTransmission THEN
                        CONTINUE;
                    ELSIF fRequestedTransmission <= fMaximumTransmission AND 
                          fRequestedTransmission >= fMinimumTransmission THEN
                        fTransmissionError := 0.0;
                    ELSE
                        fTransmissionError := fRequestedTransmission - fMinimumTransmission;
                    END_IF
                    
                    IF ABS(fTransmissionError) > ABS(fOptimalTransmissionErrorThusFar) THEN
                        CONTINUE;
                    END_IF
                    
                    fAverageTransmission := (fMaximumTransmission + fMinimumTransmission) / 2.0;
                    
                    IF ABS(fTransmissionError) = ABS(fOptimalTransmissionErrorThusFar) AND
                       ABS(fRequestedTransmission - fAverageTransmission) > ABS(fRequestedTransmission - fOptimalAverageTransmissionThusFar) THEN
                        CONTINUE;
                    END_IF
                    
                    fOptimalAverageTransmissionThusFar := fAverageTransmission;
                
                    fOptimalTransmissionErrorThusFar := fTransmissionError;
                    
                    iOptimalFilterCombination := fbFilterCombination;
                
                E_HE_SATT_RoundingMode.CLOSEST_BELOW:
                    IF fRequestedTransmission < fMinimumTransmission THEN
                        CONTINUE;
                    ELSIF fRequestedTransmission <= fMaximumTransmission AND 
                          fRequestedTransmission >= fMinimumTransmission THEN
                        fTransmissionError := 0.0;
                    ELSE
                        fTransmissionError := fRequestedTransmission - fMaximumTransmission;
                    END_IF
                    
                    IF ABS(fTransmissionError) > ABS(fOptimalTransmissionErrorThusFar) THEN
                        CONTINUE;
                    END_IF
                    
                    fAverageTransmission := (fMaximumTransmission + fMinimumTransmission) / 2.0;
                    
                    IF ABS(fTransmissionError) = ABS(fOptimalTransmissionErrorThusFar) AND
                       ABS(fRequestedTransmission - fAverageTransmission) > ABS(fRequestedTransmission - fOptimalAverageTransmissionThusFar) THEN
                        CONTINUE;
                    END_IF
                    
                    fOptimalAverageTransmissionThusFar := fAverageTransmission;
                
                    fOptimalTransmissionErrorThusFar := fTransmissionError;
                    
                    iOptimalFilterCombination := fbFilterCombination;
                    
                E_HE_SATT_RoundingMode.CLOSEST:
                    IF fRequestedTransmission > fMaximumTransmission THEN
                        fTransmissionError := fRequestedTransmission - fMaximumTransmission;
                    ELSIF fRequestedTransmission <= fMaximumTransmission AND 
                          fRequestedTransmission >= fMinimumTransmission THEN
                        fTransmissionError := 0.0;
                    ELSE
                        fTransmissionError := fRequestedTransmission - fMinimumTransmission;
                    END_IF
                    
                    IF ABS(fTransmissionError) > ABS(fOptimalTransmissionErrorThusFar) THEN
                        CONTINUE;
                    END_IF
                    
                    fAverageTransmission := (fMaximumTransmission + fMinimumTransmission) / 2.0;
                    
                    IF ABS(fTransmissionError) = ABS(fOptimalTransmissionErrorThusFar) AND
                       ABS(fRequestedTransmission - fAverageTransmission) > ABS(fRequestedTransmission - fOptimalAverageTransmissionThusFar) THEN
                        CONTINUE;
                    END_IF
                    
                    fOptimalAverageTransmissionThusFar := fAverageTransmission;
                
                    fOptimalTransmissionErrorThusFar := fTransmissionError;
                    
                    iOptimalFilterCombination := fbFilterCombination;
                    
                E_HE_SATT_RoundingMode.FIRST_ABOVE_WITHIN_TOLERANCE:
                    IF fRequestedTransmission > fMaximumTransmission THEN
                        CONTINUE;
                    ELSIF fRequestedTransmission <= fMaximumTransmission AND 
                          fRequestedTransmission >= fMinimumTransmission THEN
                        fTransmissionError := 0.0;
                    ELSE
                        fTransmissionError := fRequestedTransmission - fMinimumTransmission;
                    END_IF
                    
                    IF fTransmissionError > 0 OR ABS(fTransmissionError) > ABS(fRequestedAllowableTolerance) THEN
                        CONTINUE;
                    END_IF
                    
                    fOptimalAverageTransmissionThusFar := fAverageTransmission;
                
                    fOptimalTransmissionErrorThusFar := fTransmissionError;
                    
                    iOptimalFilterCombination := fbFilterCombination;
                    
                    RETURN;
                    
                E_HE_SATT_RoundingMode.FIRST_BELOW_WITHIN_TOLERANCE:
                    IF fRequestedTransmission < fMinimumTransmission THEN
                        CONTINUE;
                    ELSIF fRequestedTransmission <= fMaximumTransmission AND 
                          fRequestedTransmission >= fMinimumTransmission THEN
                        fTransmissionError := 0.0;
                    ELSE
                        fTransmissionError := fRequestedTransmission - fMaximumTransmission;
                    END_IF
                    
                    IF fTransmissionError < 0 OR ABS(fTransmissionError) > ABS(fRequestedAllowableTolerance) THEN
                        CONTINUE;
                    END_IF
                    
                    fOptimalAverageTransmissionThusFar := fAverageTransmission;
                
                    fOptimalTransmissionErrorThusFar := fTransmissionError;
                    
                    iOptimalFilterCombination := fbFilterCombination;
                    
                    RETURN;
                    
                E_HE_SATT_RoundingMode.FIRST_WITHIN_TOLERANCE:
                    IF fRequestedTransmission > fMaximumTransmission THEN
                        fTransmissionError := fRequestedTransmission - fMaximumTransmission;
                    ELSIF fRequestedTransmission <= fMaximumTransmission AND 
                          fRequestedTransmission >= fMinimumTransmission THEN
                        fTransmissionError := 0.0;
                    ELSE
                        fTransmissionError := fRequestedTransmission - fMinimumTransmission;
                    END_IF
                    
                    IF ABS(fTransmissionError) > ABS(fRequestedAllowableTolerance) THEN
                        CONTINUE;
                    END_IF
                    
                    fOptimalAverageTransmissionThusFar := fAverageTransmission;
                
                    fOptimalTransmissionErrorThusFar := fTransmissionError;
                    
                    iOptimalFilterCombination := fbFilterCombination;
                    
                    RETURN;
            END_CASE
        END_FOR
        
        stStatus.bBusy := FALSE;
        stStatus.bDone := TRUE;
        
        IF THIS^.iOptimalFilterCombination = 0 THEN
            stStatus.bError := TRUE;
            stStatus.sErrorMsg := 'No valid filter combination found.';
        ELSE
            stStatus.bError := FALSE;
            stStatus.sErrorMsg := '';
        END_IF
        
        eState := IDLE;
END_CASE


METHOD FB_Init: BOOL
VAR_INPUT
    bInitRetains: BOOL; // TRUE: the retain variables are initialized (reset warm / reset cold)
    bInCopyCode: BOOL;  // TRUE: the instance will be copied to the copy code afterward (online change)   
    
    iFilterCombinationToTransmission : I_HE_SATT_FilterCombinationToTransmission;
END_VAR

THIS^.iFilterCombinationToTransmission := iFilterCombinationToTransmission;
END_METHOD


METHOD PUBLIC FindOptimalCombination
VAR_INPUT
    fPhotonEnergy_eV : LREAL;
	(* [0.0 - 1.0]*)
	fRequestedTransmission	: LREAL;
	eRequestedRoundingMode	: E_HE_SATT_RoundingMode;
	fRequestedAllowableTolerance	: LREAL;
    iFilterCombinationCollector : I_HE_SATT_FilterCombinationCollector;
END_VAR
VAR_OUTPUT
    iOptimalFilterCombination : I_HE_SATT_FilterCombination;
END_VAR

THIS^.fPhotonEnergy_eV := fPhotonEnergy_eV;
THIS^.fRequestedTransmission := fRequestedTransmission;
THIS^.eRequestedRoundingMode := eRequestedRoundingMode;
THIS^.fRequestedAllowableTolerance := fRequestedAllowableTolerance;
THIS^.iFilterCombinationCollector := iFilterCombinationCollector;
    
iOptimalFilterCombination := THIS^.iOptimalFilterCombination;
END_METHOD


PROPERTY Status : REFERENCE TO ST_HE_SATT_Status
GET

Status REF= THIS^.stStatus;
END_GET
END_PROPERTY

END_FUNCTION_BLOCK

// ---- Devices/HE_SATT/FBs/FB_HE_SATT_FilterToTransmission.TcPOU

FUNCTION_BLOCK FB_HE_SATT_FilterToTransmission IMPLEMENTS I_HE_SATT_FilterToTransmission
VAR
    iScatteringFactorLookup : I_ScatteringFactorLookup;
END_VAR


METHOD PUBLIC CalculateTransmission
VAR_INPUT
    fPhotonEnergy_eV : LREAL;
    iFilter : I_HE_SATT_Filter;
END_VAR
VAR_OUTPUT
    fMinimumTransmission : LREAL;
    fMaximumTransmission : LREAL;
END_VAR
VAR    
    iFilterConstantThickness : I_HE_SATT_FilterConstantThickness;
    iFilterWedge : I_HE_SATT_FilterWedge;
    
    f2 : LREAL;
    fDensity_gm3 : LREAL;
    fAtomicWeight : LREAL;
    fMassAttenuationCoefficient : LREAL;
    
    bError : BOOL;
    sErrorMsg : T_MaxString;
END_VAR

IF iFilter = 0 THEN
    fMinimumTransmission := 1.0;
    fMaximumTransmission := fMinimumTransmission;
    RETURN;
END_IF

iScatteringFactorLookup.GetScatteringFactor(
    sMaterialName := iFilter.MaterialFormula,
    fPhotonEnergy_eV := fPhotonEnergy_eV,
    f2 => f2,
    bError => bError,
    sErrorMsg => sErrorMsg
);

IF bError THEN
    // TODO: Log error
END_IF

fDensity_gm3 := F_MaterialDensityLookup(
    sMaterialName := iFilter.MaterialFormula
) * 1e6;

fAtomicWeight := F_AtomicMassLookup(
    sMaterialName := iFilter.MaterialFormula
);

fMassAttenuationCoefficient := F_CalculateMassAttenuationCoefficient(
    f2 := f2,
    fPhotonEnergy_eV := fPhotonEnergy_eV,
    fDensity_gm3 := fDensity_gm3,
    fAtomicWeight := fAtomicWeight
);

IF __QUERYINTERFACE(iFilter, iFilterConstantThickness) THEN
    fMinimumTransmission := F_CalculateTransmission(
        fAbsorptionConstant := fMassAttenuationCoefficient,
        fThickness_in_m := iFilterConstantThickness.Thickness
    );
    
    fMaximumTransmission := fMinimumTransmission;
    
ELSIF __QUERYINTERFACE(iFilter, iFilterWedge) THEN
    fMinimumTransmission := F_CalculateTransmission(
        fAbsorptionConstant := fMassAttenuationCoefficient,
        fThickness_in_m := iFilterWedge.MaxThickness
    );
    
    fMaximumTransmission := F_CalculateTransmission(
        fAbsorptionConstant := fMassAttenuationCoefficient,
        fThickness_in_m := iFilterWedge.MinThickness
    );
ELSE
    // TODO: Log error
END_IF
END_METHOD


METHOD FB_Init: BOOL
VAR_INPUT
    bInitRetains: BOOL; // TRUE: the retain variables are initialized (reset warm / reset cold)
    bInCopyCode: BOOL;  // TRUE: the instance will be copied to the copy code afterward (online change)

    iScatteringFactorLookup : I_ScatteringFactorLookup;
END_VAR

THIS^.iScatteringFactorLookup := iScatteringFactorLookup;
END_METHOD

END_FUNCTION_BLOCK

// ---- Devices/HE_SATT/FBs/FB_HE_SATT_FilterWedge.TcPOU

FUNCTION_BLOCK FB_HE_SATT_FilterWedge EXTENDS FB_HE_SATT_Filter IMPLEMENTS I_HE_SATT_FilterWedge
VAR
    fThicknessAt0 : LREAL; // 0 is the part of the filter that is the closest to the center of the pipe when retracted.
    fThicknessAtLength : LREAL;
END_VAR


METHOD FB_Init: BOOL
VAR_INPUT
    bInitRetains: BOOL; // TRUE: the retain variables are initialized (reset warm / reset cold)
    bInCopyCode: BOOL;  // TRUE: the instance will be copied to the copy code afterward (online change)   
    
    iHolder : I_HE_SATT_FilterHolder;
    fDefaultLength : LREAL;
    eDefaultMaterial : E_HE_SATT_FilterMaterial;
    eDefaultStatus : E_HE_SATT_FilterStatus;
    fDefaultThicknessAt0 : LREAL;
    fDefaultThicknessAtLength : LREAL;
END_VAR

THIS^.iHolder := iHolder;
THIS^.fLength := fDefaultLength;
THIS^.eMaterial := eDefaultMaterial;
THIS^.eStatus := eDefaultStatus;
THIS^.fThicknessAt0 := fDefaultThicknessAt0;
THIS^.fThicknessAtLength := fDefaultThicknessAtLength;

THIS^.iHolder.RegisterFilter(THIS^);
END_METHOD


PROPERTY MaxThickness : LREAL
GET

MaxThickness := MAX(THIS^.fThicknessAt0, THIS^.fThicknessAtLength);
END_GET
END_PROPERTY


PROPERTY MinThickness : LREAL
GET

MinThickness := MIN(THIS^.fThicknessAt0, THIS^.fThicknessAtLength);
END_GET
END_PROPERTY


METHOD ThicknessAt : LREAL
VAR_INPUT
	(* Position in units of property Length and with value from 0 to value of property Length*)
	fPosition	: LREAL;
END_VAR
END_METHOD

END_FUNCTION_BLOCK

// ---- Devices/HE_SATT/FBs/FB_HE_SATT_Sequence.TcPOU

FUNCTION_BLOCK FB_HE_SATT_Sequence IMPLEMENTS I_HE_SATT_Sequence
VAR
    iFilterCombinationFinder : I_HE_SATT_FilterCombinationFinder;
    iFilterHolderSelector : I_HE_SATT_FilterHolderSelector;
    iPhotonEnergy_eV : I_HE_SATT_PhotonEnergy_eV;
    iFindOptimalFilterCombination : I_HE_SATT_FindOptimalFilterCombination;
    iFindOptimalThicknessFromFilterCombination : I_HE_SATT_FindOptimalThicknessFromFilterCombination;
    iCommands : I_HE_SATT_Commands;
    aiFilterHolder : REFERENCE TO ARRAY[1..PL_HE_SATT_Parameters.nNumHolders] OF I_HE_SATT_FilterHolder;

    eSequenceState : E_HE_SATT_SequenceState;
    
	fRequestedTransmission	: LREAL;
	eRequestedRoundingMode	: E_HE_SATT_RoundingMode;
	fRequestedAllowableTolerance	: LREAL;
    
    fbFilterCombinationCollector : FB_HE_SATT_FilterCombinationCollector;
    fbFilterCombinationCollectorDownselected : FB_HE_SATT_FilterCombinationCollector;
    
    iOptimalFilterCombination : I_HE_SATT_FilterCombination;
    
    afThickness : ARRAY[1..PL_HE_SATT_Parameters.nNumHolders] OF LREAL;
    
    nIteratorHolder : INT;
    iFilter : I_HE_SATT_Filter;
    
    bAllDone : BOOL;
END_VAR


IF iCommands.Reset THEN
    eSequenceState := E_HE_SATT_SequenceState.IDLE;
END_IF

CASE SequenceState OF
    E_HE_SATT_SequenceState.IDLE:
        // Do nothing for now
        
    E_HE_SATT_SequenceState.TRIGGER_DETERMINE_FILTER_COMBINATIONS:
        iFilterCombinationFinder.DetermineFilterCombinations(
            iFilterHolderSelector := iFilterHolderSelector,
            iFilterCombinationCollector := fbFilterCombinationCollector
        );
        
        eSequenceState := E_HE_SATT_SequenceState.CONFIRM_DETERMINE_FILTER_COMBINATIONS;
        
    E_HE_SATT_SequenceState.CONFIRM_DETERMINE_FILTER_COMBINATIONS:
        IF iFilterCombinationFinder.Status.bError THEN
            eSequenceState := E_HE_SATT_SequenceState.ERROR;
            // TODO: error handling
            RETURN;
        END_IF
        
        IF iFilterCombinationFinder.Status.bDone THEN
            eSequenceState := E_HE_SATT_SequenceState.TRIGGER_DOWNSELECT_FILTER_COMBINATIONS;
        END_IF
        
    E_HE_SATT_SequenceState.TRIGGER_DOWNSELECT_FILTER_COMBINATIONS:
        fbFilterCombinationCollector.DownselectByCouplingRule(
            iFilterHolderSelector := iFilterHolderSelector,
            iFilterCombinationCollector := fbFilterCombinationCollectorDownselected
        );
        
        eSequenceState := E_HE_SATT_SequenceState.CONFIRM_DOWNSELECT_FILTER_COMBINATIONS;
        
    E_HE_SATT_SequenceState.CONFIRM_DOWNSELECT_FILTER_COMBINATIONS:
        IF fbFilterCombinationCollector.DownselectStatus.bError THEN
            eSequenceState := E_HE_SATT_SequenceState.ERROR;
            // TODO: error handling
            RETURN;
        END_IF
        
        IF fbFilterCombinationCollector.DownselectStatus.bDone THEN
            eSequenceState := E_HE_SATT_SequenceState.TRIGGER_CALCULATE_OPTIMAL_FILTER_COMBINATION;
        END_IF
        
    E_HE_SATT_SequenceState.TRIGGER_CALCULATE_OPTIMAL_FILTER_COMBINATION:
        IF iPhotonEnergy_eV.Error THEN
            eSequenceState := E_HE_SATT_SequenceState.ERROR;
            // TODO: error handling
            RETURN;
        END_IF
    
        iFindOptimalFilterCombination.FindOptimalCombination(
            fPhotonEnergy_eV := iPhotonEnergy_eV.Value,
            fRequestedTransmission := fRequestedTransmission,
            eRequestedRoundingMode := eRequestedRoundingMode,
            fRequestedAllowableTolerance := fRequestedAllowableTolerance,
            iFilterCombinationCollector := fbFilterCombinationCollectorDownselected,
            iOptimalFilterCombination => iOptimalFilterCombination,
        );
        
        eSequenceState := E_HE_SATT_SequenceState.CONFIRM_CALCULATE_OPTIMAL_FILTER_COMBINATION;
        
    E_HE_SATT_SequenceState.CONFIRM_CALCULATE_OPTIMAL_FILTER_COMBINATION:
        IF iFindOptimalFilterCombination.Status.bError THEN
            eSequenceState := E_HE_SATT_SequenceState.ERROR;
            // TODO: error handling
            RETURN;
        END_IF
        
        IF iFindOptimalFilterCombination.Status.bDone THEN
            eSequenceState := E_HE_SATT_SequenceState.TRIGGER_CALCULATE_OPTIMAL_WEDGE_THICKNESSES;
        END_IF
        
    E_HE_SATT_SequenceState.TRIGGER_CALCULATE_OPTIMAL_WEDGE_THICKNESSES:
        IF iOptimalFilterCombination = 0 THEN
            eSequenceState := E_HE_SATT_SequenceState.ERROR;
            // TODO: error handling
            RETURN;
        END_IF
        
        IF iPhotonEnergy_eV.Error THEN
            eSequenceState := E_HE_SATT_SequenceState.ERROR;
            // TODO: error handling
            RETURN;
        END_IF
        
        iFindOptimalThicknessFromFilterCombination.FindOptimalThicknessFromFilterCombination(
            fPhotonEnergy_eV := iPhotonEnergy_eV.Value,
            fRequestedTransmission := fRequestedTransmission,
            iFilterCombination := iOptimalFilterCombination,
            afThickness => afThickness
        );
        
    E_HE_SATT_SequenceState.CONFIRM_CALCULATE_OPTIMAL_WEDGE_THICKNESSES:
        IF iFindOptimalThicknessFromFilterCombination.Status.bError THEN
            eSequenceState := E_HE_SATT_SequenceState.ERROR;
            // TODO: error handling
            RETURN;
        END_IF
        
        IF iFindOptimalThicknessFromFilterCombination.Status.bDone THEN
            eSequenceState := E_HE_SATT_SequenceState.CONFIRM_MOVE_PERMITTED;
        END_IF
        
    E_HE_SATT_SequenceState.CONFIRM_MOVE_PERMITTED:
        IF iCommands.PermitMove THEN
            eSequenceState := E_HE_SATT_SequenceState.TRIGGER_MOVE_START;
        END_IF
        
    E_HE_SATT_SequenceState.TRIGGER_MOVE_START:
        FOR nIteratorHolder := 1 TO PL_HE_SATT_Parameters.nNumHolders BY 1 DO
            iFilter := iOptimalFilterCombination.GetFilter(nIteratorHolder);
            
            aiFilterHolder[nIteratorHolder].MoveToFilter(
                iFilter := iFilter,
                fThickness := afThickness[nIteratorHolder]
            );
        END_FOR
        
        eSequenceState := E_HE_SATT_SequenceState.CONFIRM_MOVE_COMPLETE;
        
    E_HE_SATT_SequenceState.CONFIRM_MOVE_COMPLETE:
        FOR nIteratorHolder := 1 TO PL_HE_SATT_Parameters.nNumHolders BY 1 DO
            IF aiFilterHolder[nIteratorHolder].Status.bError THEN
                eSequenceState := E_HE_SATT_SequenceState.ERROR;
                // TODO: error handling
                RETURN;
            END_IF
        END_FOR
        
        bAllDone := TRUE;
        
        FOR nIteratorHolder := 1 TO PL_HE_SATT_Parameters.nNumHolders BY 1 DO
            bAllDone := bAllDone AND aiFilterHolder[nIteratorHolder].Status.bDone;
        END_FOR
        
        IF bAllDone THEN
            eSequenceState := E_HE_SATT_SequenceState.IDLE;
            // TODO: lof successful completion of move.
        END_IF
        
    E_HE_SATT_SequenceState.ERROR:
        // TODO: error handling
        
END_CASE


METHOD FB_Init: BOOL
VAR_INPUT
    bInitRetains: BOOL; // TRUE: the retain variables are initialized (reset warm / reset cold)
    bInCopyCode: BOOL;  // TRUE: the instance will be copied to the copy code afterward (online change)   
    
    iFilterCombinationFinder : I_HE_SATT_FilterCombinationFinder;
    iFilterHolderSelector : I_HE_SATT_FilterHolderSelector;
    iFindOptimalFilterCombination : I_HE_SATT_FindOptimalFilterCombination;
    iPhotonEnergy_eV : I_HE_SATT_PhotonEnergy_eV;
    iCommands : I_HE_SATT_Commands;
    aiFilterHolder : REFERENCE TO ARRAY[1..PL_HE_SATT_Parameters.nNumHolders] OF I_HE_SATT_FilterHolder;
END_VAR

THIS^.iFilterCombinationFinder := iFilterCombinationFinder;
THIS^.iFilterHolderSelector := iFilterHolderSelector;
THIS^.iFindOptimalFilterCombination := iFindOptimalFilterCombination;
THIS^.iPhotonEnergy_eV := iPhotonEnergy_eV;
THIS^.iCommands := iCommands;
THIS^.aiFilterHolder REf= aiFilterHolder;
END_METHOD

PROPERTY PUBLIC SequenceState : E_HE_SATT_SequenceState
GET

SequenceState := THIS^.eSequenceState;
END_GET
END_PROPERTY


METHOD Start
VAR_INPUT
	(* [0.0 - 1.0]*)
	fRequestedTransmission	: LREAL;
	eRequestedRoundingMode	: E_HE_SATT_RoundingMode;
	fRequestedAllowableTolerance	: LREAL;
END_VAR

THIS^.fRequestedTransmission := fRequestedTransmission;
THIS^.eRequestedRoundingMode := eRequestedRoundingMode;
THIS^.fRequestedAllowableTolerance := fRequestedAllowableTolerance;

THIS^.eSequenceState := E_HE_SATT_SequenceState.TRIGGER_DETERMINE_FILTER_COMBINATIONS;
END_METHOD

END_FUNCTION_BLOCK

// ---- Devices/HE_SATT/FBs/FB_HE_SATT_UserRequest.TcPOU

FUNCTION_BLOCK FB_HE_SATT_UserRequest
VAR
    iHE_SATT_Sequence : I_HE_SATT_Sequence;

    fRequestedTransmission : LREAL; // [0.0 - 1.0] - Link to epics read-write
    fRequestedTransmissionAfterInputValidation : LREAL; // [0.0 - 1.0] - Link to epics but read only
    eRequestedRoundingMode : E_HE_SATT_RoundingMode; // Link to epics read-write
    eRequestedRoundingModeAfterInputValidation : E_HE_SATT_RoundingMode; // Link to epics but read-only
    fRequestedAllowableTolerance : LREAL; // Link to epics read-write
    fRequestedAllowableToleranceAfterInputValidation : LREAL; // Link to epics but read-only
    
    bApplyConfig : BOOL; // Link to epics - read-write
END_VAR


IF bApplyConfig THEN
    ApplyConfig();
    bApplyConfig := FALSE;
END_IF


METHOD PUBLIC ApplyConfig

IF NOT IsFinite(x := F_LREAL(THIS^.fRequestedTransmission)) OR NOT IsFinite(x := F_LREAL(THIS^.fRequestedAllowableTolerance)) THEN
    RETURN;
END_IF

CASE THIS^.eRequestedRoundingMode OF
    E_HE_SATT_RoundingMode.CLOSEST_ABOVE:
        THIS^.eRequestedRoundingModeAfterInputValidation := THIS^.eRequestedRoundingMode;
        
    E_HE_SATT_RoundingMode.FIRST_ABOVE_WITHIN_TOLERANCE:
        THIS^.eRequestedRoundingModeAfterInputValidation := THIS^.eRequestedRoundingMode;
        
    E_HE_SATT_RoundingMode.CLOSEST_BELOW:
        THIS^.eRequestedRoundingModeAfterInputValidation := THIS^.eRequestedRoundingMode;
        
    E_HE_SATT_RoundingMode.FIRST_BELOW_WITHIN_TOLERANCE:
        THIS^.eRequestedRoundingModeAfterInputValidation := THIS^.eRequestedRoundingMode;
        
    E_HE_SATT_RoundingMode.CLOSEST:
        THIS^.eRequestedRoundingModeAfterInputValidation := THIS^.eRequestedRoundingMode;
        
    E_HE_SATT_RoundingMode.FIRST_WITHIN_TOLERANCE:
        THIS^.eRequestedRoundingModeAfterInputValidation := THIS^.eRequestedRoundingMode;
        
    ELSE
        THIS^.eRequestedRoundingModeAfterInputValidation := E_HE_SATT_RoundingMode.FIRST_BELOW_WITHIN_TOLERANCE;
END_CASE

THIS^.fRequestedTransmissionAfterInputValidation := LIMIT(0.0, THIS^.fRequestedTransmission, 1.0);

THIS^.fRequestedAllowableToleranceAfterInputValidation := LIMIT(0.0, THIS^.fRequestedAllowableTolerance, 1.0);

THIS^.iHE_SATT_Sequence.Start(
    fRequestedTransmission := THIS^.fRequestedTransmissionAfterInputValidation,
    eRequestedRoundingMode := THIS^.eRequestedRoundingModeAfterInputValidation,
    fRequestedAllowableTolerance := THIS^.fRequestedAllowableToleranceAfterInputValidation
);
END_METHOD


METHOD FB_Init: BOOL
VAR_INPUT
    bInitRetains: BOOL; // TRUE: the retain variables are initialized (reset warm / reset cold)
    bInCopyCode: BOOL;  // TRUE: the instance will be copied to the copy code afterward (online change)
    
    iHE_SATT_Sequence : I_HE_SATT_Sequence;
END_VAR

THIS^.iHE_SATT_Sequence := iHE_SATT_Sequence;
END_METHOD


METHOD PUBLIC RequestTransmission
VAR_INPUT
    fRequestedTransmission : LREAL; // [0.0 - 1.0]
    eRequestedRoundingMode : E_HE_SATT_RoundingMode;
    fRequestedAllowableTolerance : LREAL;
END_VAR

THIS^.fRequestedTransmission := fRequestedTransmission;
THIS^.eRequestedRoundingMode := eRequestedRoundingMode;
THIS^.fRequestedAllowableTolerance := fRequestedAllowableTolerance;
END_METHOD

END_FUNCTION_BLOCK

// ---- Devices/PPM/FB_PPM_PowerMeter.TcPOU
FUNCTION_BLOCK FB_PPM_PowerMeter
VAR_INPUT
    fTempSP: REAL;
    bVetoTempFFO: BOOL;
    sDeviceName: STRING;

    // Used to know when to stop background auto-collection
    eEnumGet: E_PPM_States;
    stYAxisState: DWORD;

    // Calibrated for each gentec, should be passed as input
    // If not set, responsive energy will not be calculated
    {attribute 'pytmc' := '
        pv: RESP
        io: i
        field: EGU V/W
    '}
    fResponsivity: LREAL;

    // Passed to FB_AnalogInput
    // The initial values are correct for EL3062,
    // but not for EL3602, which needs iTermBits:=31
    // with fTermMax and fTermMin dependent on what
    // range the terminal was configured to use
    // (default -10000mV to +10000mV)
    iTermBits : UINT := 15;
    fTermMax : REAL := 10000;
    fTermMin: REAL := 0;
END_VAR
VAR_IN_OUT
    fbFFHWO: FB_HardwareFFOutput;
END_VAR
VAR
    iVoltageINT AT %I*: DINT;

    {attribute 'pytmc' := '
        pv: VOLT
        io: input
        field: EGU mV
    '}
    fVoltage: LREAL;

    {attribute 'pytmc' := '
        pv: VOLT_BUFFER
        io: input
        field: EGU mV
    '}
    fVoltageBuffer: ARRAY[1..1000] OF LREAL;

    {attribute 'pytmc' := '
        pv: STC
        io: input
    '}
    fbTempSensor: FB_CC_TempSensor;


    fFrequency: REAL;
    // Used to get beam rate
    {attribute 'pytmc' := '
        pv: SXR_NC_BeamRateFromEpics
        link: EVNT:SYS0:1:NC_SOFTRATE
    '}
    fSXR_NC_Frequency: REAL;
    {attribute 'pytmc' := '
        pv: SXR_SC_BeamRateFromEpics
        link: TPG:SYS0:1:DST04:RATE_RBV
    '}
    uSXR_SC_Frequency: UINT;

    {attribute 'pytmc' := '
        pv: HXR_NC_BeamRateFromEpics
        link: EVNT:SYS0:1:NC_HARDRATE
    '}
    fHXR_NC_Frequency: REAL;
    {attribute 'pytmc' := '
        pv: HXR_SC_BeamRateFromEpics
        link: TPG:SYS0:1:DST03:RATE_RBV
    '}
    uHXR_SC_Frequency: UINT;

    // Pulse-by-pulse energy and buffer
    {attribute 'pytmc' := '
        pv: MJ
        io: i
        field: EGU mJ
    '}
    fCalibMJ: LREAL;
    {attribute 'pytmc' := '
        pv: MJ_BUFFER
        io: i
        field: EGU mJ
    '}
    fCalibMJBuffer: ARRAY[1..1000] OF LREAL;

    // Wattage and buffer
    {attribute 'pytmc' := '
        pv: WATT
        io: i
        field: EGU mW
    '}
    fPulseWattage: LREAL;
    {attribute 'pytmc' := '
        pv: WATT_BUFFER
        io: i
        field: EGU mW
    '}
    fPulseWattageBuffer: ARRAY[1..1000] OF LREAL;

    // Background voltage
    {attribute 'pytmc' := '
        pv: BACK:VOLT
        io: io
        field: EGU mV
    '}
    fBackgroundVoltage: LREAL;

    // Internal variables for background voltage auto-collection
    fBackgroundVoltageAcc: LREAL;
    uAccCount: UINT;
    fBackgroundVoltageSum: LREAL;
    fBackgroundVoltageStale: LREAL;
    tonBackgroundAutoCollecting: TON;
    fBackgroundVoltageBuffer: ARRAY[1..100] OF LREAL;
    udBackgroundVoltageBufferIndex: UDINT := 1;
    rTrig_Background : R_TRIG;
    i: UDINT;
    // Used to reset auto-collected background buffer, and fBackgroundVoltage if in Auto mode
    {attribute 'pytmc' := '
        pv: BACK:RESET
        io: io
    '}
    bResetAutoBackground: BOOL;

    // In manual mode, auto-background updates buffer but does not change fBackgroundVoltage
    {attribute 'pytmc' := '
        pv: BACK:MODE
        io: io
    '}
    BACKGROUND_MODE: (Manual, Auto) := Auto;

    // Boolean to trigger collection of background voltages
    {attribute 'pytmc' := '
        pv: BACK:COLL
        io: io
    '}
    bBackgroundCollect: BOOL;

    // Time in seconds to collect background voltages for
    {attribute 'pytmc' := '
        pv: BACK:TIME
        io: io
        field: EGU s
    '}
    uBackgroundCollectionTime: UINT := 60;
    tofBackgroundCollecting: TOF;
    udBackgroundManualCount: UDINT;
    // Boolean indicating when background is being manually collected
    {attribute 'pytmc' := '
        pv: BACK:MANUAL_COLLECTING
        io: i
    '}
    bBackgroundCollecting: BOOL := FALSE;

    fbGetPMVoltage: FB_AnalogInput;

    fbVoltageBuffer: FB_LREALBuffer;
    fbPulseWattageBuffer: FB_LREALBuffer;
    fbCalibMJBuffer: FB_LREALBuffer;
END_VAR

fbTempSensor(
    fFaultThreshold:=fTempSP,
    bVeto:=bVetoTempFFO,
    sDevName:=sDeviceName,
    io_fbFFHWO:=fbFFHWO,
);

// Convert the terminal's integer into a value in millivolts
// If you get a compile-time error about converting type DINT
// to type INT, update your lcls-general version to at least
// v2.12.0
fbGetPMVoltage(
    iRaw := TO_INT(iVoltageINT),
    iTermBits := iTermBits,
    fTermMax := fTermMax,
    fTermMin := fTermMin,
    fReal => fVoltage);

rTrig_Background(CLK:=(eEnumGet <> E_PPM_States.OUT OR stYAxisState <> 0));
// Reset buffer and related variables
IF rTrig_Background.Q OR bResetAutoBackground THEN
    IF bResetAutoBackground THEN
        bResetAutoBackground := FALSE;
        IF BACKGROUND_MODE = Auto THEN
            fBackgroundVoltage := 0;
        END_IF
    ELSE
        // Dump 5s worth of readings
        IF udBackgroundVoltageBufferIndex > 6 THEN
            FOR i := (udBackgroundVoltageBufferIndex - 5) TO (udBackgroundVoltageBufferIndex - 1) DO
                fBackgroundVoltageSum := fBackgroundVoltageSum - fBackgroundVoltageBuffer[((i-1) MOD 100) + 1];
            END_FOR
            udBackgroundVoltageBufferIndex := udBackgroundVoltageBufferIndex - 5;
            IF udBackgroundVoltageBufferIndex <> 1 AND BACKGROUND_MODE = Auto THEN
                fBackgroundVoltage := fBackgroundVoltageSum / MIN((udBackgroundVoltageBufferIndex - 1), 100);
            END_IF
        ELSIF BACKGROUND_MODE = Auto THEN
                fBackgroundVoltage := 0;
        END_IF
    END_IF
    fBackgroundVoltageAcc := 0;
    fBackgroundVoltageSum := 0;
    tonBackgroundAutoCollecting(IN := FALSE);
    udBackgroundVoltageBufferIndex := 1;
ELSIF eEnumGet = E_PPM_States.OUT AND stYAxisState = 0 THEN
    tonBackgroundAutoCollecting( IN := TRUE, PT := T#1000MS);
    // Every second, move fBackgroundVoltageAcc into buffer and sum
    IF tonBackgroundAutoCollecting.Q = TRUE THEN
        tonBackgroundAutoCollecting( IN := FALSE);
        fBackgroundVoltageStale := fBackgroundVoltageBuffer[((udBackgroundVoltageBufferIndex - 1) MOD 100) + 1];
        fBackgroundVoltageBuffer[((udBackgroundVoltageBufferIndex - 1) MOD 100) + 1] := fBackgroundVoltageAcc / uAccCount;
        // Remove overwritten voltage
        IF udBackgroundVoltageBufferIndex > 100 THEN
            fBackgroundVoltageSum := fBackgroundVoltageSum - fBackgroundVoltageStale;
        END_IF
        fBackgroundVoltageSum := fBackgroundVoltageSum + fBackgroundVoltageAcc / uAccCount;
        fBackgroundVoltageAcc := fVoltage;
        uAccCount := 1;
        udBackgroundVoltageBufferIndex := udBackgroundVoltageBufferIndex + 1;
    ELSE
        uAccCount := uAccCount + 1;
        fBackgroundVoltageAcc := fBackgroundVoltageAcc + fVoltage;
    END_IF

END_IF

IF udBackgroundVoltageBufferIndex <> 1 AND BACKGROUND_MODE = Auto THEN
    fBackgroundVoltage := fBackgroundVoltageSum / MIN((udBackgroundVoltageBufferIndex - 1), 100);
END_IF

// Start collecting background in manual mode - 60s by default but can be set with uBackgroundCollectionTime
IF bBackgroundCollect = TRUE AND BACKGROUND_MODE = Manual THEN
    bBackgroundCollect := FALSE;
    udBackgroundManualCount := 0;
    fBackgroundVoltage := 0;
    tofBackgroundCollecting(IN := TRUE);
END_IF

bBackgroundCollecting := FALSE;
tofBackgroundCollecting(IN := FALSE, PT := UINT_TO_TIME(uBackgroundCollectionTime * 1000));
IF tofBackgroundCollecting.Q = TRUE THEN
    IF BACKGROUND_MODE = Manual THEN
        bBackgroundCollecting := TRUE;
        udBackgroundManualCount := udBackgroundManualCount + 1;
        fBackgroundVoltage := (fBackgroundVoltage * (udBackgroundManualCount - 1) + fVoltage) / udBackgroundManualCount;
    END_IF
END_IF

// Getting frequency based on accelerator source
{IF defined (K)}
    IF PMPS_GVL.stCurrentBeamParameters.nMachineMode = 0 THEN
        fFrequency := fSXR_NC_Frequency;
    ELSIF PMPS_GVL.stCurrentBeamParameters.nMachineMode = 1 THEN
        fFrequency := uSXR_SC_Frequency;
    END_IF
{ELSIF defined (L)}
    IF PMPS_GVL.stCurrentBeamParameters.nMachineMode = 0 THEN
        fFrequency := fHXR_NC_Frequency;
    ELSIF PMPS_GVL.stCurrentBeamParameters.nMachineMode = 1 THEN
        fFrequency := uHXR_SC_Frequency;
    END_IF
{END_IF}

// Getting wattage and energy
fPulseWattage := SEL(fResponsivity <> 0, 0, (fVoltage - fBackgroundVoltage) / fResponsivity);
fCalibMJ := SEL(fFrequency <> 0, -9999, fPulseWattage / fFrequency);

// Buffer the full-rate Voltage, Pulse wattage, and calibrated MJ values
fbVoltageBuffer(
    bExecute := TRUE,
    fInput := fVoltage,
    arrOutput => fVoltageBuffer);
fbPulseWattageBuffer(
    bExecute := TRUE,
    fInput := fPulseWattage,
    arrOutput => fPulseWattageBuffer);
fbCalibMJBuffer(
    bExecute := TRUE,
    fInput := fCalibMJ,
    arrOutput => fCalibMJBuffer);

END_FUNCTION_BLOCK

// ---- Tests/HE_SATT/FB_HE_SATT_EpicsHeartBeat_Test.TcPOU

FUNCTION_BLOCK FB_HE_SATT_EpicsHeartBeat_Test EXTENDS FB_TestSuite


GivenThatHeartbeatIsProvidedExpectNoExpiration();
GivenThatHeartbeatTimeHasExpiredExpectHeartBeatPropertyToIndicateSo();


METHOD PRIVATE GivenThatHeartbeatIsProvidedExpectNoExpiration
VAR_INST
    fbTestTimer : TON := (PT := T#2S, IN := TRUE);

    // Subject under test
    fbHE_SATT_EpicsHeartBeat : FB_HE_SATT_EpicsHeartBeat(tTimeout := T#1S);
END_VAR

TEST('GivenThatHeartbeatIsProvidedExpectNoExpiration');

fbTestTimer();
fbHE_SATT_EpicsHeartBeat.Heartbeat();
fbHE_SATT_EpicsHeartBeat();

IF fbTestTimer.Q THEN
    AssertFalse(Condition := fbHE_SATT_EpicsHeartBeat.IsHeartbeatExpired(),
                Message := 'Expected heart beat to expire');
    TEST_FINISHED();
END_IF
END_METHOD


METHOD PRIVATE GivenThatHeartbeatTimeHasExpiredExpectHeartBeatPropertyToIndicateSo
VAR_INST
    fbTestTimer : TON := (PT := T#2S, IN := TRUE);

    // Subject under test
    fbHE_SATT_EpicsHeartBeat : FB_HE_SATT_EpicsHeartBeat(tTimeout := T#1S);
END_VAR

TEST('GivenThatHeartbeatTimeHasExpiredExpectHeartBeatPropertyToIndicateSo');

fbTestTimer();
fbHE_SATT_EpicsHeartBeat();

IF fbTestTimer.Q THEN
    AssertTrue(Condition := fbHE_SATT_EpicsHeartBeat.IsHeartbeatExpired(),
               Message := 'Expected heart beat to expire');
    TEST_FINISHED();
END_IF
END_METHOD

END_FUNCTION_BLOCK

// ---- Tests/HE_SATT/FB_HE_SATT_FilterCombinationCollector_Test.TcPOU

FUNCTION_BLOCK FB_HE_SATT_FilterCombinationCollector_Test EXTENDS FB_TestSuite


GivenCouplingExpectCorrectDownselectedListOfCombinations();


METHOD PRIVATE AssertEquals_Combination
VAR_INPUT
    iFilterCombinationExpected : I_HE_SATT_FilterCombination;
    iFilterCombinationResult : I_HE_SATT_FilterCombination;
END_VAR
VAR
    sMessageBuilder : T_MaxString;
    nIteratorHolder : INT;
    iFilterExpected : I_HE_SATT_Filter;
    iFilterResult : I_HE_SATT_Filter;
END_VAR

FOR nIteratorHolder := 1 TO PL_HE_SATT_Parameters.nNumHolders BY 1 DO
    iFilterExpected := iFilterCombinationExpected.GetFilter(nIteratorHolder);
    iFilterResult := iFilterCombinationResult.GetFilter(nIteratorHolder);
    sMessageBuilder := 'Combination filter in slot for holder ';
    sMessageBuilder := CONCAT(sMessageBuilder, TO_STRING(nIteratorHolder));
    sMessageBuilder := CONCAT(sMessageBuilder, ' was not the expected filter. ');
    AssertTrue(
        Condition := iFilterExpected = iFilterResult,
        Message := sMessageBuilder
    );
END_FOR
END_METHOD


METHOD PRIVATE GivenCouplingExpectCorrectDownselectedListOfCombinations
VAR
    afbFilter : ARRAY[1..PL_HE_SATT_Parameters.nNumHolders] OF FB_HE_SATT_FilterTestDouble;    
    
    fbFilterHolderSelector : FB_HE_SATT_FilterHolderSelector;

    // Subject under test
    fbFilterCombinationCollector1 : FB_HE_SATT_FilterCombinationCollector;
    fbFilterCombinationCollector2 : FB_HE_SATT_FilterCombinationCollector;

    // Variables for test
    sConcatString : T_MaxString;
    fbFilterCombination : FB_HE_SATT_FilterCombination;
    fbFilterCombinationExpected : FB_HE_SATT_FilterCombination;
    aiFilterExpected : ARRAY[1..PL_HE_SATT_Parameters.nNumHolders] OF I_HE_SATT_Filter;
    fbFilterCombinationResult : FB_HE_SATT_FilterCombination;
    aiFilterResult : ARRAY[1..PL_HE_SATT_Parameters.nNumHolders] OF I_HE_SATT_Filter;
    abCoupledHolders : ARRAY[1..PL_HE_SATT_Parameters.nNumHolders] OF BOOL;
END_VAR

TEST('GivenCouplingExpectCorrectDownselectedListOfCombinations');

// Couple 3 and 4 so that they must always be used together.
abCoupledHolders[3] := abCoupledHolders[4] := TRUE;

fbFilterHolderSelector.CoupleHolders(abCoupledHolders);

fbFilterCombinationCollector2.Reset();

fbFilterCombination.Clear();

// Add a filter combination that doesn't use any filters.
fbFilterCombinationCollector1.AddFilterCombination(fbFilterCombination);

// Downselect should pick up the combination that doesn't use any filters.
fbFilterCombinationCollector1.DownselectByCouplingRule(
    iFilterCombinationCollector := fbFilterCombinationCollector2,
    iFilterHolderSelector := fbFilterHolderSelector
);

AssertEquals_DINT(
    Expected := 1,
    Actual := fbFilterCombinationCollector2.NumCombinationsAdded,
    Message := 'Number of combinations found was not correct.'
);

fbFilterCombinationExpected.Clear();
fbFilterCombinationResult := fbFilterCombinationCollector2.GetCombination(1);
AssertEquals_Combination(
    iFilterCombinationExpected := fbFilterCombinationExpected,
    iFilterCombinationResult := fbFilterCombinationResult
);

fbFilterCombinationCollector2.Reset();

// Add a combination that only uses filter 3.
fbFilterCombination.Clear();
fbFilterCombination.AddFilter(3, afbFilter[3]);

fbFilterCombinationCollector1.AddFilterCombination(fbFilterCombination);

// Downselect by 3 to 4 coupling means this combination should be filtered out of the result.
fbFilterCombinationCollector1.DownselectByCouplingRule(
    iFilterCombinationCollector := fbFilterCombinationCollector2,
    iFilterHolderSelector := fbFilterHolderSelector
);

AssertEquals_DINT(
    Expected := 1,
    Actual := fbFilterCombinationCollector2.NumCombinationsAdded,
    Message := 'Number of combinations found was not correct.'
);

fbFilterCombinationCollector2.Reset();

// Now we add 3 and 4 and the downselected result should contain this combination.
fbFilterCombination.Clear();
fbFilterCombination.AddFilter(3, afbFilter[3]);
fbFilterCombination.AddFilter(4, afbFilter[4]);

fbFilterCombinationCollector1.AddFilterCombination(fbFilterCombination);

fbFilterCombinationCollector1.DownselectByCouplingRule(
    iFilterCombinationCollector := fbFilterCombinationCollector2,
    iFilterHolderSelector := fbFilterHolderSelector
);

AssertEquals_DINT(
    Expected := 2,
    Actual := fbFilterCombinationCollector2.NumCombinationsAdded,
    Message := 'Number of combinations found was not correct.'
);

fbFilterCombinationExpected.Clear();
fbFilterCombinationExpected.AddFilter(1, 0);
fbFilterCombinationExpected.AddFilter(2, 0);
fbFilterCombinationExpected.AddFilter(3, afbFilter[3]);
fbFilterCombinationExpected.AddFilter(4, afbFilter[4]);
fbFilterCombinationExpected.AddFilter(5, 0);
fbFilterCombinationResult := fbFilterCombinationCollector2.GetCombination(2);
AssertEquals_Combination(
    iFilterCombinationExpected := fbFilterCombinationExpected,
    iFilterCombinationResult := fbFilterCombinationResult
);

fbFilterCombinationExpected.Clear();
fbFilterCombinationResult := fbFilterCombinationCollector2.GetCombination(3);
AssertEquals_Combination(
    iFilterCombinationExpected := fbFilterCombinationExpected,
    iFilterCombinationResult := fbFilterCombinationResult
);

TEST_FINISHED();
END_METHOD

END_FUNCTION_BLOCK

// ---- Tests/Test Doubles/FB_HE_SATT_FilterTestDouble.TcPOU

FUNCTION_BLOCK FB_HE_SATT_FilterTestDouble IMPLEMENTS I_HE_SATT_Filter
VAR
    iHolder : I_HE_SATT_FilterHolder;
    fLength : LREAL;
    eMaterial : E_HE_SATT_FilterMaterial;
    fPositionInHolder : LREAL;
    eStatus : E_HE_SATT_FilterStatus;
END_VAR


PROPERTY Holder : I_HE_SATT_FilterHolder
GET

Holder := THIS^.iHolder;
END_GET
SET

THIS^.iHolder := Holder;
END_SET
END_PROPERTY


PROPERTY Length : LREAL
GET

Length := THIS^.fLength;
END_GET
SET

THIS^.fLength := Length;
END_SET
END_PROPERTY


PROPERTY Material : E_HE_SATT_FilterMaterial
GET

Material := THIS^.eMaterial;
END_GET
SET

THIS^.eMaterial := Material;
END_SET
END_PROPERTY


PROPERTY PositionInHolder : LREAL
GET

PositionInHolder := THIS^.fPositionInHolder;
END_GET
SET

THIS^.fPositionInHolder := PositionInHolder;
END_SET
END_PROPERTY


PROPERTY Status : E_HE_SATT_FilterStatus
GET

Status := THIS^.eStatus;
END_GET
SET

THIS^.eStatus := Status;
END_SET
END_PROPERTY

END_FUNCTION_BLOCK

// ---- Tests/HE_SATT/FB_HE_SATT_FindOptimalFilterCombination_Test.TcPOU

FUNCTION_BLOCK FB_HE_SATT_FindOptimalFilterCombination_Test EXTENDS FB_TestSuite
VAR
    nAssertEquals_CombinationCounter : INT;
END_VAR


GivenCombinationCollectionAndRequestExpectOptimalCombinationFound();


METHOD PRIVATE AssertEquals_Combination
VAR_INPUT
    iFilterCombinationExpected : I_HE_SATT_FilterCombination;
    iFilterCombinationResult : I_HE_SATT_FilterCombination;
END_VAR
VAR
    sMessageBuilder : T_MaxString;
    nIteratorHolder : INT;
    iFilterExpected : I_HE_SATT_Filter;
    iFilterResult : I_HE_SATT_Filter;
END_VAR

nAssertEquals_CombinationCounter := nAssertEquals_CombinationCounter + 1;

FOR nIteratorHolder := 1 TO PL_HE_SATT_Parameters.nNumHolders BY 1 DO
    iFilterExpected := iFilterCombinationExpected.GetFilter(nIteratorHolder);
    iFilterResult := iFilterCombinationResult.GetFilter(nIteratorHolder);
    sMessageBuilder := 'Combination filter in slot for holder ';
    sMessageBuilder := CONCAT(sMessageBuilder, TO_STRING(nIteratorHolder));
    sMessageBuilder := CONCAT(sMessageBuilder, ' was not the expected filter. ');
    sMessageBuilder := CONCAT(sMessageBuilder, '# ');
    sMessageBuilder := CONCAT(sMessageBuilder, TO_STRING(nAssertEquals_CombinationCounter));
    AssertTrue(
        Condition := iFilterExpected = iFilterResult,
        Message := sMessageBuilder
    );
END_FOR
END_METHOD


METHOD PRIVATE GivenCombinationCollectionAndRequestExpectOptimalCombinationFound
VAR
    // Test fixture
    afbFilter : ARRAY[1..PL_HE_SATT_Parameters.nNumHolders] OF FB_HE_SATT_FilterTestDouble;    
    
    fbFilterCombination : FB_HE_SATT_FilterCombination;
    
    fbFilterCombinationCollector : FB_HE_SATT_FilterCombinationCollector;
    
    fbFilterCombinationToTransmissionTestDouble : FB_HE_SATT_FilterCombinationToTransmissionTestDouble;

    // Subject under test
    fbHE_SATT_FindOptimalFilterCombination : FB_HE_SATT_FindOptimalFilterCombination(
        iFilterCombinationToTransmission := fbFilterCombinationToTransmissionTestDouble
    );

    // Variables for test
    sConcatString : T_MaxString;
    fbFilterCombinationExpected : FB_HE_SATT_FilterCombination;
    aiFilterExpected : ARRAY[1..PL_HE_SATT_Parameters.nNumHolders] OF I_HE_SATT_Filter;
    iFilterCombinationResult : I_HE_SATT_FilterCombination;
    aiFilterResult : ARRAY[1..PL_HE_SATT_Parameters.nNumHolders] OF I_HE_SATT_Filter;
END_VAR

TEST('GivenCombinationCollectionAndRequestExpectOptimalCombinationFound');

fbFilterCombination.Clear();
fbFilterCombinationToTransmissionTestDouble.PushTransmissionResultToSequence(
    fMinimumTransmission := 1.0,
    fMaximumTransmission := 1.0
);
fbFilterCombinationCollector.AddFilterCombination(fbFilterCombination);

fbFilterCombination.Clear();
fbFilterCombination.AddFilter(1, afbFilter[1]);
fbFilterCombinationToTransmissionTestDouble.PushTransmissionResultToSequence(
    fMinimumTransmission := 0.8,
    fMaximumTransmission := 0.8
);
fbFilterCombinationCollector.AddFilterCombination(fbFilterCombination);

fbFilterCombination.Clear();
fbFilterCombination.AddFilter(1, afbFilter[1]);
fbFilterCombination.AddFilter(2, afbFilter[2]);
fbFilterCombinationToTransmissionTestDouble.PushTransmissionResultToSequence(
    fMinimumTransmission := 0.7,
    fMaximumTransmission := 0.7
);
fbFilterCombinationCollector.AddFilterCombination(fbFilterCombination);

fbFilterCombination.Clear();
fbFilterCombination.AddFilter(3, afbFilter[3]);
fbFilterCombination.AddFilter(4, afbFilter[4]);
fbFilterCombinationToTransmissionTestDouble.PushTransmissionResultToSequence(
    fMinimumTransmission := 0.6,
    fMaximumTransmission := 0.8
);
fbFilterCombinationCollector.AddFilterCombination(fbFilterCombination);

fbFilterCombination.Clear();
fbFilterCombination.AddFilter(1, afbFilter[1]);
fbFilterCombination.AddFilter(2, afbFilter[2]);
fbFilterCombination.AddFilter(5, afbFilter[5]);
fbFilterCombinationToTransmissionTestDouble.PushTransmissionResultToSequence(
    fMinimumTransmission := 0.1,
    fMaximumTransmission := 0.9
);
fbFilterCombinationCollector.AddFilterCombination(fbFilterCombination);

fbFilterCombination.Clear();
fbFilterCombination.AddFilter(1, afbFilter[1]);
fbFilterCombination.AddFilter(3, afbFilter[3]);
fbFilterCombination.AddFilter(5, afbFilter[5]);
fbFilterCombinationToTransmissionTestDouble.PushTransmissionResultToSequence(
    fMinimumTransmission := 0.95,
    fMaximumTransmission := 0.95
);
fbFilterCombinationCollector.AddFilterCombination(fbFilterCombination);

fbHE_SATT_FindOptimalFilterCombination.FindOptimalCombination(
    fPhotonEnergy_eV := 1000,
    fRequestedTransmission := 0.61,
    eRequestedRoundingMode := E_HE_SATT_RoundingMode.CLOSEST_ABOVE,
    fRequestedAllowableTolerance := 1e-3,
    iFilterCombinationCollector := fbFilterCombinationCollector,
    iOptimalFilterCombination => iFilterCombinationResult
);

fbFilterCombinationExpected.Clear();
fbFilterCombinationExpected.AddFilter(1, 0);
fbFilterCombinationExpected.AddFilter(2, 0);
fbFilterCombinationExpected.AddFilter(3, afbFilter[3]);
fbFilterCombinationExpected.AddFilter(4, afbFilter[4]);
fbFilterCombinationExpected.AddFilter(5, 0);
AssertEquals_Combination(
    iFilterCombinationExpected := fbFilterCombinationExpected,
    iFilterCombinationResult := iFilterCombinationResult
);

fbFilterCombinationToTransmissionTestDouble.Reset();

fbHE_SATT_FindOptimalFilterCombination.FindOptimalCombination(
    fPhotonEnergy_eV := 1000,
    fRequestedTransmission := 0.94,
    eRequestedRoundingMode := E_HE_SATT_RoundingMode.CLOSEST_BELOW,
    fRequestedAllowableTolerance := 1e-3,
    iFilterCombinationCollector := fbFilterCombinationCollector,
    iOptimalFilterCombination => iFilterCombinationResult
);

fbFilterCombinationExpected.Clear();
fbFilterCombinationExpected.AddFilter(1, afbFilter[1]);
fbFilterCombinationExpected.AddFilter(2, afbFilter[2]);
fbFilterCombinationExpected.AddFilter(3, 0);
fbFilterCombinationExpected.AddFilter(4, 0);
fbFilterCombinationExpected.AddFilter(5, afbFilter[5]);
AssertEquals_Combination(
    iFilterCombinationExpected := fbFilterCombinationExpected,
    iFilterCombinationResult := iFilterCombinationResult
);

fbFilterCombinationToTransmissionTestDouble.Reset();

fbHE_SATT_FindOptimalFilterCombination.FindOptimalCombination(
    fPhotonEnergy_eV := 1000,
    fRequestedTransmission := 0.96,
    eRequestedRoundingMode := E_HE_SATT_RoundingMode.CLOSEST,
    fRequestedAllowableTolerance := 1e-3,
    iFilterCombinationCollector := fbFilterCombinationCollector,
    iOptimalFilterCombination => iFilterCombinationResult
);

fbFilterCombinationExpected.Clear();
fbFilterCombinationExpected.AddFilter(1, afbFilter[1]);
fbFilterCombinationExpected.AddFilter(2, 0);
fbFilterCombinationExpected.AddFilter(3, afbFilter[3]);
fbFilterCombinationExpected.AddFilter(4, 0);
fbFilterCombinationExpected.AddFilter(5, afbFilter[5]);
AssertEquals_Combination(
    iFilterCombinationExpected := fbFilterCombinationExpected,
    iFilterCombinationResult := iFilterCombinationResult
);

fbFilterCombinationToTransmissionTestDouble.Reset();

fbHE_SATT_FindOptimalFilterCombination.FindOptimalCombination(
    fPhotonEnergy_eV := 1000,
    fRequestedTransmission := 0.79,
    eRequestedRoundingMode := E_HE_SATT_RoundingMode.FIRST_ABOVE_WITHIN_TOLERANCE,
    fRequestedAllowableTolerance := 0.02,
    iFilterCombinationCollector := fbFilterCombinationCollector,
    iOptimalFilterCombination => iFilterCombinationResult
);

fbFilterCombinationExpected.Clear();
fbFilterCombinationExpected.AddFilter(1, afbFilter[1]);
fbFilterCombinationExpected.AddFilter(2, 0);
fbFilterCombinationExpected.AddFilter(3, 0);
fbFilterCombinationExpected.AddFilter(4, 0);
fbFilterCombinationExpected.AddFilter(5, 0);
AssertEquals_Combination(
    iFilterCombinationExpected := fbFilterCombinationExpected,
    iFilterCombinationResult := iFilterCombinationResult
);

fbFilterCombinationToTransmissionTestDouble.Reset();

fbHE_SATT_FindOptimalFilterCombination.FindOptimalCombination(
    fPhotonEnergy_eV := 1000,
    fRequestedTransmission := 0.79,
    eRequestedRoundingMode := E_HE_SATT_RoundingMode.FIRST_BELOW_WITHIN_TOLERANCE,
    fRequestedAllowableTolerance := 0.1,
    iFilterCombinationCollector := fbFilterCombinationCollector,
    iOptimalFilterCombination => iFilterCombinationResult
);

fbFilterCombinationExpected.Clear();
fbFilterCombinationExpected.AddFilter(1, afbFilter[1]);
fbFilterCombinationExpected.AddFilter(2, afbFilter[2]);
fbFilterCombinationExpected.AddFilter(3, 0);
fbFilterCombinationExpected.AddFilter(4, 0);
fbFilterCombinationExpected.AddFilter(5, 0);
AssertEquals_Combination(
    iFilterCombinationExpected := fbFilterCombinationExpected,
    iFilterCombinationResult := iFilterCombinationResult
);

fbFilterCombinationToTransmissionTestDouble.Reset();

fbHE_SATT_FindOptimalFilterCombination.FindOptimalCombination(
    fPhotonEnergy_eV := 1000,
    fRequestedTransmission := 0.89,
    eRequestedRoundingMode := E_HE_SATT_RoundingMode.FIRST_WITHIN_TOLERANCE,
    fRequestedAllowableTolerance := 0.1,
    iFilterCombinationCollector := fbFilterCombinationCollector,
    iOptimalFilterCombination => iFilterCombinationResult
);

fbFilterCombinationExpected.Clear();
fbFilterCombinationExpected.AddFilter(1, afbFilter[1]);
fbFilterCombinationExpected.AddFilter(2, 0);
fbFilterCombinationExpected.AddFilter(3, 0);
fbFilterCombinationExpected.AddFilter(4, 0);
fbFilterCombinationExpected.AddFilter(5, 0);
AssertEquals_Combination(
    iFilterCombinationExpected := fbFilterCombinationExpected,
    iFilterCombinationResult := iFilterCombinationResult
);

fbFilterCombinationToTransmissionTestDouble.Reset();

fbHE_SATT_FindOptimalFilterCombination.FindOptimalCombination(
    fPhotonEnergy_eV := 1000,
    fRequestedTransmission := 0.55,
    eRequestedRoundingMode := E_HE_SATT_RoundingMode.FIRST_WITHIN_TOLERANCE,
    fRequestedAllowableTolerance := 0.1,
    iFilterCombinationCollector := fbFilterCombinationCollector,
    iOptimalFilterCombination => iFilterCombinationResult
);

fbFilterCombinationExpected.Clear();
fbFilterCombinationExpected.AddFilter(1, 0);
fbFilterCombinationExpected.AddFilter(2, 0);
fbFilterCombinationExpected.AddFilter(3, afbFilter[3]);
fbFilterCombinationExpected.AddFilter(4, afbFilter[4]);
fbFilterCombinationExpected.AddFilter(5, 0);
AssertEquals_Combination(
    iFilterCombinationExpected := fbFilterCombinationExpected,
    iFilterCombinationResult := iFilterCombinationResult
);

fbFilterCombinationToTransmissionTestDouble.Reset();

TEST_FINISHED();
END_METHOD

END_FUNCTION_BLOCK

// ---- Tests/Test Doubles/FB_HE_SATT_FilterCombinationToTransmissionTestDouble.TcPOU

FUNCTION_BLOCK FB_HE_SATT_FilterCombinationToTransmissionTestDouble IMPLEMENTS I_HE_SATT_FilterCombinationToTransmission
VAR CONSTANT
    nMaxIndex : INT := 10;
END_VAR
VAR
    afMinimumTransmissionResultSequence : ARRAY[1..nMaxIndex] OF LREAL;
    afMaximumTransmissionResultSequence : ARRAY[1..nMaxIndex] OF LREAL;
    nIndexForNextAdditionToSequence : INT;
    nIndexInSequence : INT;
END_VAR


METHOD CalculateTransmission
VAR_INPUT
	fPhotonEnergy_eV	: LREAL;
	iFilterCombination	: I_HE_SATT_FilterCombination;
END_VAR
VAR_OUTPUT
	fMinimumTransmission	: LREAL;
	fMaximumTransmission	: LREAL;
END_VAR

THIS^.nIndexInSequence := THIS^.nIndexInSequence + 1;

fMinimumTransmission := THIS^.afMinimumTransmissionResultSequence[THIS^.nIndexInSequence];
fMaximumTransmission := THIS^.afMaximumTransmissionResultSequence[THIS^.nIndexInSequence];

IF THIS^.nIndexInSequence > THIS^.nMaxIndex THEN
    THIS^.nIndexInSequence := 0;
END_IF
END_METHOD


METHOD PUBLIC PushTransmissionResultToSequence
VAR_INPUT
    fMinimumTransmission : LREAL;
    fMaximumTransmission : LREAL;
END_VAR

THIS^.nIndexForNextAdditionToSequence := THIS^.nIndexForNextAdditionToSequence + 1;

THIS^.afMinimumTransmissionResultSequence[THIS^.nIndexForNextAdditionToSequence] := fMinimumTransmission;
THIS^.afMaximumTransmissionResultSequence[THIS^.nIndexForNextAdditionToSequence] := fMaximumTransmission;
END_METHOD


METHOD PUBLIC Reset

THIS^.nIndexInSequence := 0;
END_METHOD

END_FUNCTION_BLOCK

// ---- Tests/HE_SATT/FB_HE_SATT_FilterHolderSelector_Test.TcPOU

FUNCTION_BLOCK FB_HE_SATT_FilterHolderSelector_Test EXTENDS FB_TestSuite


GivenCoupledHoldersExpectCorrectFiltering_1();
GivenCoupledHoldersExpectCorrectFiltering_2();


METHOD PRIVATE GivenCoupledHoldersExpectCorrectFiltering_1
VAR_INST
    // Test fixture   
    afbFilterTestDouble : ARRAY[1..PL_HE_SATT_Parameters.nNumHolders] OF FB_HE_SATT_FilterTestDouble;
 
    fbFilterCombination : FB_HE_SATT_FilterCombination;

    // Subject under test
    fbFilterHolderSelector : FB_HE_SATT_FilterHolderSelector;
    
    // Variables for test
    abCoupledHolders : ARRAY[1..PL_HE_SATT_Parameters.nNumHolders] OF BOOL;
    bExpected : BOOL;
    bResult : BOOL;
END_VAR

TEST('GivenCoupledHoldersExpectCorrectFiltering_1');

fbFilterCombination.AddFilter(1, afbFilterTestDouble[1]);
fbFilterCombination.AddFilter(2, afbFilterTestDouble[2]);
fbFilterCombination.AddFilter(4, afbFilterTestDouble[4]);

abCoupledHolders[1] := abCoupledHolders[2] := abCoupledHolders[3] := TRUE;

fbFilterHolderSelector.CoupleHolders(abCoupledHolders);

bExpected := FALSE;

bResult := fbFilterHolderSelector.CouplingRulesSatisfied(
    iFilterCombination := fbFilterCombination
);

AssertEquals_BOOL(
    Expected := bExpected,
    Actual := bResult,
    Message := 'Expected coupling rules to not be satisfied.'
);

fbFilterCombination.AddFilter(3, afbFilterTestDouble[3]);

bExpected := TRUE;

bResult := fbFilterHolderSelector.CouplingRulesSatisfied(
    iFilterCombination := fbFilterCombination
);

AssertEquals_BOOL(
    Expected := bExpected,
    Actual := bResult,
    Message := 'Expected coupling rules to be satisfied.'
);

TEST_FINISHED();
END_METHOD


METHOD PRIVATE GivenCoupledHoldersExpectCorrectFiltering_2
VAR_INST
    // Test fixture   
    afbFilterTestDouble : ARRAY[1..PL_HE_SATT_Parameters.nNumHolders] OF FB_HE_SATT_FilterTestDouble;
 
    fbFilterCombination : FB_HE_SATT_FilterCombination;

    // Subject under test
    fbFilterHolderSelector : FB_HE_SATT_FilterHolderSelector;
    
    // Variables for test
    abCoupledHolders : ARRAY[1..PL_HE_SATT_Parameters.nNumHolders] OF BOOL;
    bExpected : BOOL;
    bResult : BOOL;
END_VAR

TEST('GivenCoupledHoldersExpectCorrectFiltering_2');

fbFilterCombination.AddFilter(2, afbFilterTestDouble[2]);
fbFilterCombination.AddFilter(4, afbFilterTestDouble[4]);

abCoupledHolders[3] := abCoupledHolders[4] := TRUE;

fbFilterHolderSelector.CoupleHolders(abCoupledHolders);

bExpected := FALSE;

bResult := fbFilterHolderSelector.CouplingRulesSatisfied(
    iFilterCombination := fbFilterCombination
);

AssertEquals_BOOL(
    Expected := bExpected,
    Actual := bResult,
    Message := 'Expected coupling rules to not be satisfied.'
);

fbFilterCombination.AddFilter(3, afbFilterTestDouble[3]);

bExpected := TRUE;

bResult := fbFilterHolderSelector.CouplingRulesSatisfied(
    iFilterCombination := fbFilterCombination
);

AssertEquals_BOOL(
    Expected := bExpected,
    Actual := bResult,
    Message := 'Expected coupling rules to be satisfied.'
);

TEST_FINISHED();
END_METHOD

END_FUNCTION_BLOCK

// ---- Tests/HE_SATT/FB_HE_SATT_FilterCombinationFinder_Test.TcPOU

FUNCTION_BLOCK FB_HE_SATT_FilterCombinationFinder_Test EXTENDS FB_TestSuite


GivenHoldersAndSelectionExpectCorrectListOfCombinations();


METHOD PRIVATE AssertEquals_Combination
VAR_INPUT
    iFilterCombinationExpected : I_HE_SATT_FilterCombination;
    iFilterCombinationResult : I_HE_SATT_FilterCombination;
END_VAR
VAR
    sMessageBuilder : T_MaxString;
    nIteratorHolder : INT;
    iFilterExpected : I_HE_SATT_Filter;
    iFilterResult : I_HE_SATT_Filter;
END_VAR

FOR nIteratorHolder := 1 TO PL_HE_SATT_Parameters.nNumHolders BY 1 DO
    iFilterExpected := iFilterCombinationExpected.GetFilter(nIteratorHolder);
    iFilterResult := iFilterCombinationResult.GetFilter(nIteratorHolder);
    sMessageBuilder := 'Combination filter in slot for holder ';
    sMessageBuilder := CONCAT(sMessageBuilder, TO_STRING(nIteratorHolder));
    sMessageBuilder := CONCAT(sMessageBuilder, ' was not the expected filter. ');
    AssertTrue(
        Condition := iFilterExpected = iFilterResult,
        Message := sMessageBuilder
    );
END_FOR
END_METHOD


METHOD PRIVATE GivenHoldersAndSelectionExpectCorrectListOfCombinations
VAR
    fbFilterHolderTestDouble : ARRAY[1..PL_HE_SATT_Parameters.nNumHolders] OF FB_HE_SATT_FilterHolderTestDouble;
    
    aiFilterHolder : ARRAY[1..PL_HE_SATT_Parameters.nNumHolders] OF I_HE_SATT_FilterHolder := [
        fbFilterHolderTestDouble[1],
        fbFilterHolderTestDouble[2],
        fbFilterHolderTestDouble[3],
        fbFilterHolderTestDouble[4],
        fbFilterHolderTestDouble[5]
    ];
    
    afbFilter : ARRAY[1..13] OF FB_HE_SATT_FilterTestDouble := [
        (Holder := fbFilterHolderTestDouble[1], Status := E_HE_SATT_FilterStatus.ENABLED),
        (Holder := fbFilterHolderTestDouble[1], Status := E_HE_SATT_FilterStatus.ENABLED),
        (Holder := fbFilterHolderTestDouble[1], Status := E_HE_SATT_FilterStatus.ENABLED),
        (Holder := fbFilterHolderTestDouble[2], Status := E_HE_SATT_FilterStatus.ENABLED),
        (Holder := fbFilterHolderTestDouble[2], Status := E_HE_SATT_FilterStatus.ENABLED),
        (Holder := fbFilterHolderTestDouble[3], Status := E_HE_SATT_FilterStatus.ENABLED),
        (Holder := fbFilterHolderTestDouble[3], Status := E_HE_SATT_FilterStatus.DISABLED),
        (Holder := fbFilterHolderTestDouble[3], Status := E_HE_SATT_FilterStatus.ENABLED),
        (Holder := fbFilterHolderTestDouble[3], Status := E_HE_SATT_FilterStatus.ENABLED),
        (Holder := fbFilterHolderTestDouble[4], Status := E_HE_SATT_FilterStatus.ENABLED),
        (Holder := fbFilterHolderTestDouble[4], Status := E_HE_SATT_FilterStatus.DISABLED),
        (Holder := fbFilterHolderTestDouble[5], Status := E_HE_SATT_FilterStatus.ENABLED),
        (Holder := fbFilterHolderTestDouble[5], Status := E_HE_SATT_FilterStatus.ENABLED)
    ];    
    
    fbFilterCombinationCollector : FB_HE_SATT_FilterCombinationCollector;
    
    fbFilterHolderSelectorTestDouble : FB_HE_SATT_FilterHolderSelectorTestDouble;

    // Subject under test
    fbFilterCombinationFinder : FB_HE_SATT_FilterCombinationFinder(
        aiFilterHolder := aiFilterHolder,
        nMaxNumberOfCombinationsFoundPerCycle := 500
    );

    // Variables for test
    sConcatString : T_MaxString;
    fbFilterCombinationExpected : FB_HE_SATT_FilterCombination;
    aiFilterExpected : ARRAY[1..PL_HE_SATT_Parameters.nNumHolders] OF I_HE_SATT_Filter;
    fbFilterCombinationResult : FB_HE_SATT_FilterCombination;
    aiFilterResult : ARRAY[1..PL_HE_SATT_Parameters.nNumHolders] OF I_HE_SATT_Filter;
END_VAR

TEST('GivenHoldersAndSelectionExpectCorrectListOfCombinations');

fbFilterHolderTestDouble[1].SetFilter(1, afbFilter[1]);
fbFilterHolderTestDouble[1].SetFilter(2, afbFilter[2]);
fbFilterHolderTestDouble[1].SetFilter(3, afbFilter[3]);
fbFilterHolderTestDouble[1].NumberOfSlots := 3;

fbFilterHolderTestDouble[2].SetFilter(1, afbFilter[4]);
fbFilterHolderTestDouble[2].SetFilter(2, afbFilter[5]);
fbFilterHolderTestDouble[2].NumberOfSlots := 2;

fbFilterHolderTestDouble[3].SetFilter(1, afbFilter[6]);
fbFilterHolderTestDouble[3].SetFilter(2, afbFilter[7]);
fbFilterHolderTestDouble[3].SetFilter(3, afbFilter[8]);
fbFilterHolderTestDouble[3].SetFilter(4, afbFilter[9]);
fbFilterHolderTestDouble[3].NumberOfSlots := 4;

fbFilterHolderTestDouble[4].SetFilter(1, afbFilter[10]);
fbFilterHolderTestDouble[4].SetFilter(2, afbFilter[11]);
fbFilterHolderTestDouble[4].NumberOfSlots := 2;

fbFilterHolderTestDouble[5].SetFilter(1, afbFilter[12]);
fbFilterHolderTestDouble[5].SetFilter(2, afbFilter[13]);
fbFilterHolderTestDouble[5].NumberOfSlots := 2;

fbFilterHolderSelectorTestDouble.DeselectHolder(1);
fbFilterHolderSelectorTestDouble.SelectHolder(2);
fbFilterHolderSelectorTestDouble.SelectHolder(3);
fbFilterHolderSelectorTestDouble.SelectHolder(4);
fbFilterHolderSelectorTestDouble.DeselectHolder(5);

fbFilterCombinationFinder.DetermineFilterCombinations(
    iFilterHolderSelector := fbFilterHolderSelectorTestDouble,
    iFilterCombinationCollector := fbFilterCombinationCollector
);

AssertEquals_BOOL(
    Expected := TRUE,
    Actual := fbFilterCombinationFinder.Status.bBusy,
    Message := 'bBusy bit should be true after calling determine filter combinations.'
);

AssertEquals_BOOL(
    Expected := FALSE,
    Actual := fbFilterCombinationFinder.Status.bDone,
    Message := 'bDone bit should be false after calling determine filter combinations.'
);

AssertEquals_BOOL(
    Expected := FALSE,
    Actual := fbFilterCombinationFinder.Status.bError,
    Message := 'bError bit should be false after calling determine filter combinations.'
);

AssertEquals_STRING(
    Expected := '',
    Actual := fbFilterCombinationFinder.Status.sErrorMsg,
    Message := 'sErrorMsg string should be emptry after calling determine filter combinations.'
);

fbFilterCombinationFinder();

AssertEquals_BOOL(
    Expected := FALSE,
    Actual := fbFilterCombinationFinder.Status.bBusy,
    Message := 'bBusy bit should be false after first function body call since less combination than max per cycle.'
);

AssertEquals_BOOL(
    Expected := TRUE,
    Actual := fbFilterCombinationFinder.Status.bDone,
    Message := 'bDone bit should be true after first function body call since less combination than max per cycle.'
);

AssertEquals_BOOL(
    Expected := FALSE,
    Actual := fbFilterCombinationFinder.Status.bError,
    Message := 'Should have been no errors after function body call.'
);

AssertEquals_STRING(
    Expected := '',
    Actual := fbFilterCombinationFinder.Status.sErrorMsg,
    Message := 'Should have been no errors after function body call.'
);

AssertEquals_DINT(
    Expected := 24,
    Actual := fbFilterCombinationCollector.NumCombinationsAdded,
    Message := 'Number of combinations found was not correct.'
);

fbFilterCombinationExpected.Clear();
fbFilterCombinationResult := fbFilterCombinationCollector.GetCombination(1);
AssertEquals_Combination(
    iFilterCombinationExpected := fbFilterCombinationExpected,
    iFilterCombinationResult := fbFilterCombinationResult
);

fbFilterCombinationExpected.Clear();
fbFilterCombinationExpected.AddFilter(1, 0);
fbFilterCombinationExpected.AddFilter(2, afbFilter[4]);
fbFilterCombinationExpected.AddFilter(3, 0);
fbFilterCombinationExpected.AddFilter(4, 0);
fbFilterCombinationExpected.AddFilter(5, 0);
fbFilterCombinationResult := fbFilterCombinationCollector.GetCombination(2);
AssertEquals_Combination(
    iFilterCombinationExpected := fbFilterCombinationExpected,
    iFilterCombinationResult := fbFilterCombinationResult
);

fbFilterCombinationExpected.Clear();
fbFilterCombinationExpected.AddFilter(1, 0);
fbFilterCombinationExpected.AddFilter(2, afbFilter[4]);
fbFilterCombinationExpected.AddFilter(3, afbFilter[8]);
fbFilterCombinationExpected.AddFilter(4, 0);
fbFilterCombinationExpected.AddFilter(5, 0);
fbFilterCombinationResult := fbFilterCombinationCollector.GetCombination(8);
AssertEquals_Combination(
    iFilterCombinationExpected := fbFilterCombinationExpected,
    iFilterCombinationResult := fbFilterCombinationResult
);

fbFilterCombinationExpected.Clear();
fbFilterCombinationExpected.AddFilter(1, 0);
fbFilterCombinationExpected.AddFilter(2, afbFilter[4]);
fbFilterCombinationExpected.AddFilter(3, afbFilter[8]);
fbFilterCombinationExpected.AddFilter(4, afbFilter[10]);
fbFilterCombinationExpected.AddFilter(5, 0);
fbFilterCombinationResult := fbFilterCombinationCollector.GetCombination(20);
AssertEquals_Combination(
    iFilterCombinationExpected := fbFilterCombinationExpected,
    iFilterCombinationResult := fbFilterCombinationResult
);

fbFilterCombinationExpected.Clear();
fbFilterCombinationExpected.AddFilter(1, 0);
fbFilterCombinationExpected.AddFilter(2, afbFilter[5]);
fbFilterCombinationExpected.AddFilter(3, afbFilter[9]);
fbFilterCombinationExpected.AddFilter(4, afbFilter[10]);
fbFilterCombinationExpected.AddFilter(5, 0);
fbFilterCombinationResult := fbFilterCombinationCollector.GetCombination(24);
AssertEquals_Combination(
    iFilterCombinationExpected := fbFilterCombinationExpected,
    iFilterCombinationResult := fbFilterCombinationResult
);

fbFilterCombinationExpected.Clear();
fbFilterCombinationResult := fbFilterCombinationCollector.GetCombination(25);
AssertEquals_Combination(
    iFilterCombinationExpected := fbFilterCombinationExpected,
    iFilterCombinationResult := fbFilterCombinationResult
);

TEST_FINISHED();
END_METHOD

END_FUNCTION_BLOCK

// ---- Tests/Test Doubles/FB_HE_SATT_FilterHolderTestDouble.TcPOU

FUNCTION_BLOCK FB_HE_SATT_FilterHolderTestDouble IMPLEMENTS I_HE_SATT_FilterHolder
VAR
    nNumberOfSlots : INT;
    aiFilter : ARRAY[1..PL_HE_SATT_Parameters.nMaxNumFiltersPerHolder] Of I_HE_SATT_Filter;
END_VAR


METHOD PUBLIC GetFilter : I_HE_SATT_Filter
VAR_INPUT
	nFilterNumber	: INT;
END_VAR

